Assert.ThatBool(
	actual := _List.Empty,
	message := "Clear with release must empty the list"
).IsTrue();

IF _UseDynamicStorage THEN
	Assert.ThatBool(
		actual := _List.Capacity = 0 AND_THEN GetBufferAddress() = TOF_Core.Memory.NULL_ADDRESS,
		message := "Clear with release must drop the dynamic allocation"
	).IsTrue();
ELSE
	Assert.ThatBool(
		actual := _List.Capacity = 12 AND_THEN GetBufferAddress() = buffer,
		message := "Clear with release must preserve the inline allocation"
	).IsTrue();
END_IF
END_METHOD

//! <summary>Borrows the concrete class name. Callers must not modify it.</summary>
{attribute 'monitoring' := 'call'}
PROPERTY ClassName : REFERENCE TO STRING
GET
ClassName REF= _ClassName;
END_GET
END_PROPERTY

//! <summary>Borrows the compiler-initialized namespace name. Callers must not modify it.</summary>
{attribute 'monitoring' := 'call'}
PROPERTY NamespaceName : REFERENCE TO STRING
GET
NamespaceName REF= CurrentNamespace.Name;
END_GET
END_PROPERTY

//! <summary>Reports the concrete instance size in bytes.</summary>
{attribute 'monitoring' := 'call'}
PROPERTY SelfSize : ULINT
GET
SelfSize := XSIZEOF(THIS^);
END_GET
END_PROPERTY

END_FUNCTION_BLOCK

// ---- Tests/Collections/Static/StaticByteListTestGroup.TcPOU
(*
SPDX-FileCopyrightText: c 2026 Oleksandr Tiutyk <trofimich@gmail.com>
SPDX-License-Identifier: MIT
License: https://opensource.org/license/mit
*)

(*!
<summary>Groups fixed-capacity byte-list operations and overflow handling.</summary>
<description>
Owns the independent child instances and their fixed registration array. Use from one PLC task at a stable address.
</description>
*)

{attribute 'no_assign'}
{attribute 'no_explicit_call' := 'do not call this function block directly'}
FUNCTION_BLOCK StaticByteListTestGroup EXTENDS TOF_Testing.TestGroup<7>
VAR_STAT
	{attribute 'hide'}
	_ClassName : STRING := __POUNAME();
END_VAR
VAR
	_LoadFromAny : ByteListLoadFromAnyTest(name := "LoadFromAny", parent := THIS^, useDynamicStorage := FALSE);
	_GetAndSet : ByteListIndexedAccessTest(name := "GetAndSet", parent := THIS^, useDynamicStorage := FALSE);
	_Find : ByteListFindTest(name := "Find", parent := THIS^, useDynamicStorage := FALSE);
	_Remove : ByteListRemoveValueTest(name := "Remove", parent := THIS^, useDynamicStorage := FALSE);
	_RemoveAt : ByteListRemoveRangeTest(name := "RemoveAt", parent := THIS^, useDynamicStorage := FALSE);
	_Clear : ByteListClearTest(name := "Clear", parent := THIS^, useDynamicStorage := FALSE);
	_Overflow : StaticByteListOverflowTest(name := "Overflow", parent := THIS^);

	_Children : ARRAY [0.._ChildCount - 1] OF TOF_Testing.ITestElement :=
	[
		_LoadFromAny,
		_GetAndSet,
		_Find,
		_Remove,
		_RemoveAt,
		_Clear,
		_Overflow
	];
END_VAR

//! <summary>Borrows the fixed child array. Callers must not modify it.</summary>
{attribute 'monitoring' := 'call'}
PROPERTY Children : REFERENCE TO ARRAY [0.._ChildCount - 1] OF TOF_Testing.ITestElement
GET
Children REF= _Children;
END_GET
END_PROPERTY

//! <summary>Borrows the concrete class name. Callers must not modify it.</summary>
{attribute 'monitoring' := 'call'}
PROPERTY ClassName : REFERENCE TO STRING
GET
ClassName REF= _ClassName;
END_GET
END_PROPERTY

//! <summary>Borrows the compiler-initialized namespace name. Callers must not modify it.</summary>
{attribute 'monitoring' := 'call'}
PROPERTY NamespaceName : REFERENCE TO STRING
GET
NamespaceName REF= CurrentNamespace.Name;
END_GET
END_PROPERTY

//! <summary>Reports the concrete instance size in bytes.</summary>
{attribute 'monitoring' := 'call'}
PROPERTY SelfSize : ULINT
GET
SelfSize := XSIZEOF(THIS^);
END_GET
END_PROPERTY

END_FUNCTION_BLOCK

// ---- Tests/Collections/Static/StaticByteListOverflowTest.TcPOU
(*
SPDX-FileCopyrightText: c 2026 Oleksandr Tiutyk <trofimich@gmail.com>
SPDX-License-Identifier: MIT
License: https://opensource.org/license/mit
*)

(*!
<summary>Checks full-capacity rejection, unchanged bytes and subsequent reuse.</summary>
<description>
Owns a fixed-capacity byte list. Run from one task at a stable address. Teardown clears the logical bytes.
</description>
*)

{attribute 'no_assign'}
{attribute 'no_explicit_call' := 'do not call this function block directly'}
FUNCTION_BLOCK StaticByteListOverflowTest EXTENDS TOF_Testing.SingleCycleTest
VAR_STAT
	{attribute 'hide'}
	_ClassName : STRING := __POUNAME();
END_VAR
VAR
	_List : TOF_Collections.ByteList<12>;
END_VAR

(*!
<summary>Checks full-capacity rejection, unchanged bytes and subsequent reuse.</summary>
*)
METHOD PROTECTED ExecuteTest
VAR
	values : ARRAY [0..11] OF BYTE := [1, 2, 3, 4, 5, 6, 7, 8, 9, 10, 11, 12];
	i : DINT;

	exceptionCode : __SYSTEM.ExceptionCode;
	caught : TOF_Core.IException;
	fullException : TOF_Core.IStaticCollectionFullException;
END_VAR
_List.AppendAny(data := values);

Assert.ThatBool(
	actual := _List.Full AND_THEN _List.Length = 12 AND_THEN _List.Capacity = 12,
	message := "The list must accept exactly twelve bytes"
).IsTrue();

__TRY
	_List.AppendByte(value := BYTE#255);
__CATCH(exceptionCode)
	caught := TOF_Core.ExceptionManager.GetLastException(
		exceptionCode := exceptionCode,
		catchPointNamespaceName := NamespaceName,
		catchPointPOUName := __POUNAME(),
		catchPointPosition := __POSITION()
	);
__ENDTRY

Assert.ThatBool(
	actual := __QUERYINTERFACE(caught, fullException),
	message := "Appending to a full list must raise StaticCollectionFullException"
).IsTrue();

Assert.ThatBool(
	actual := _List.Full AND_THEN _List.Length = 12 AND_THEN _List.Capacity = 12,
	message := "Rejected append must preserve the full list and its capacity"
).IsTrue();

FOR i := 0 TO 11 DO
	Assert.ThatByte(
		actual := _List.Get(index := i),
		message := "Rejected append must preserve every byte"
	).ToBe(expected := values[i]);
END_FOR

_List.RemoveAt(index := 11, count := 1);
_List.AppendByte(value := BYTE#255);

Assert.ThatBool(
	actual := _List.Full AND_THEN _List.Get(index := 11) = BYTE#255,
	message := "Freeing one slot must allow the next append"
).IsTrue();
END_METHOD

(*!
<summary>Restores the fixture before the runner publishes the result.</summary>
<description>
Also runs after an unexpected exception interrupts the case.
</description>
*)
METHOD PROTECTED AfterTest
_List.Clear(releaseDynamicMemory := TRUE);
END_METHOD

//! <summary>Borrows the concrete class name. Callers must not modify it.</summary>
{attribute 'monitoring' := 'call'}
PROPERTY ClassName : REFERENCE TO STRING
GET
ClassName REF= _ClassName;
END_GET
END_PROPERTY

//! <summary>Borrows the compiler-initialized namespace name. Callers must not modify it.</summary>
{attribute 'monitoring' := 'call'}
PROPERTY NamespaceName : REFERENCE TO STRING
GET
NamespaceName REF= CurrentNamespace.Name;
END_GET
END_PROPERTY

//! <summary>Reports the concrete instance size in bytes.</summary>
{attribute 'monitoring' := 'call'}
PROPERTY SelfSize : ULINT
GET
SelfSize := XSIZEOF(THIS^);
END_GET
END_PROPERTY

END_FUNCTION_BLOCK

// ---- Tests/JSON/AutomaticJsonSerializerTestGroup.TcPOU
(*
SPDX-FileCopyrightText: c 2026 Oleksandr Tiutyk <trofimich@gmail.com>
SPDX-License-Identifier: MIT
License: https://opensource.org/license/mit
*)

(*!
<summary>Groups native JSON conversion, capacity, encoding and callback cases.</summary>
<description>
Owns the independent child instances and their fixed registration array. Use from one PLC task at a stable address.
</description>
*)

{attribute 'no_assign'}
{attribute 'no_explicit_call' := 'do not call this function block directly'}
FUNCTION_BLOCK AutomaticJsonSerializerTestGroup EXTENDS TOF_Testing.TestGroup<12>
VAR_STAT
	{attribute 'hide'}
	_ClassName : STRING := __POUNAME();
END_VAR
VAR
	_RoundTripsAnyStructure : AutomaticJsonRoundTripsAnyStructureTest(name := "RoundTripsAnyStructure", parent := THIS^);
	_ThrowingAnyRoundTrip : AutomaticJsonThrowingAnyRoundTripTest(name := "ThrowingAnyRoundTrip", parent := THIS^);
	_SingleFieldVarInfoRoundTrip : AutomaticJsonSingleFieldVarInfoRoundTripTest(name := "SingleFieldVarInfoRoundTrip", parent := THIS^);
	_RejectsInvalidArguments : AutomaticJsonRejectsInvalidArgumentsTest(name := "RejectsInvalidArguments", parent := THIS^);
	_ThrowingArgumentCategories : AutomaticJsonThrowingArgumentCategoriesTest(name := "ThrowingArgumentCategories", parent := THIS^);
	_MalformedJsonAndReuse : AutomaticJsonMalformedJsonAndReuseTest(name := "MalformedJsonAndReuse", parent := THIS^);
	_WrappedCallbacks : AutomaticJsonWrappedCallbacksTest(name := "WrappedCallbacks", parent := THIS^);
	_CallbackContainmentAndReuse : AutomaticJsonCallbackContainmentAndReuseTest(name := "CallbackContainmentAndReuse", parent := THIS^);
	_ThrowingCallbackPropagation : AutomaticJsonThrowingCallbackPropagationTest(name := "ThrowingCallbackPropagation", parent := THIS^);
	_CapacityOverflowAndReuse : AutomaticJsonCapacityOverflowAndReuseTest(name := "CapacityOverflowAndReuse", parent := THIS^);
	_LongUtf8RoundTrip : AutomaticJsonLongUtf8RoundTripTest(name := "LongUtf8RoundTrip", parent := THIS^);
	_DecimalPlacesReadback : AutomaticJsonDecimalPlacesReadbackTest(name := "DecimalPlacesReadback", parent := THIS^);

	_Children : ARRAY [0.._ChildCount - 1] OF TOF_Testing.ITestElement :=
	[
		_RoundTripsAnyStructure,
		_ThrowingAnyRoundTrip,
		_SingleFieldVarInfoRoundTrip,
		_RejectsInvalidArguments,
		_ThrowingArgumentCategories,
		_MalformedJsonAndReuse,
		_WrappedCallbacks,
		_CallbackContainmentAndReuse,
		_ThrowingCallbackPropagation,
		_CapacityOverflowAndReuse,
		_LongUtf8RoundTrip,
		_DecimalPlacesReadback
	];
END_VAR

//! <summary>Borrows the fixed child array. Callers must not modify it.</summary>
{attribute 'monitoring' := 'call'}
PROPERTY Children : REFERENCE TO ARRAY [0.._ChildCount - 1] OF TOF_Testing.ITestElement
GET
Children REF= _Children;
END_GET
END_PROPERTY

//! <summary>Borrows the concrete class name. Callers must not modify it.</summary>
{attribute 'monitoring' := 'call'}
PROPERTY ClassName : REFERENCE TO STRING
GET
ClassName REF= _ClassName;
END_GET
END_PROPERTY

//! <summary>Borrows the compiler-initialized namespace name. Callers must not modify it.</summary>
{attribute 'monitoring' := 'call'}
PROPERTY NamespaceName : REFERENCE TO STRING
GET
NamespaceName REF= CurrentNamespace.Name;
END_GET
END_PROPERTY

//! <summary>Reports the concrete instance size in bytes.</summary>
{attribute 'monitoring' := 'call'}
PROPERTY SelfSize : ULINT
GET
SelfSize := XSIZEOF(THIS^);
END_GET
END_PROPERTY

END_FUNCTION_BLOCK

// ---- Tests/JSON/AutomaticJsonRoundTripsAnyStructureTest.TcPOU
(*
SPDX-FileCopyrightText: c 2026 Oleksandr Tiutyk <trofimich@gmail.com>
SPDX-License-Identifier: MIT
License: https://opensource.org/license/mit
*)

(*!
<summary>Checks successful ANY Try conversion and copied byte count.</summary>
<description>
Owns persistent native serializer state and any payload buffers used by this case.
Run from one task at a stable address. The caller provides task-boundary exception cleanup.
</description>
*)

{attribute 'no_assign'}
{attribute 'no_explicit_call' := 'do not call this function block directly'}
FUNCTION_BLOCK AutomaticJsonRoundTripsAnyStructureTest EXTENDS TOF_Testing.SingleCycleTest
VAR_STAT
	{attribute 'hide'}
	_ClassName : STRING := __POUNAME();
END_VAR
VAR
	_Serializer : TOF_JSON.AutomaticJsonSerializer;
	_Source : JSON_TEST_VALUE;
	_Target : JSON_TEST_VALUE;
	_Json : TOF_Core.JSON_DOCUMENT;
END_VAR

(*!
<summary>Checks successful ANY Try conversion and copied byte count.</summary>
*)
METHOD PROTECTED ExecuteTest
VAR
	success : BOOL;
	jsonSize : UDINT;
	expectedJson : STRING(40) := '{"Number":42,"Ready":true}';
END_VAR
_Source.Number := 42;
_Source.Ready := TRUE;

_Target.Number := 0;
_Target.Ready := FALSE;

_Json := '';

success := _Serializer.TrySerialize(
	sourceStructure := _Source,
	extender := 0,
	targetJson := _Json,
	jsonSize => jsonSize
);
Assert.ThatBool(
	actual := success,
	message := "ANY TryCreate must succeed"
).IsTrue();
Assert.ThatUDInt(
	actual := jsonSize,
	message := "Copy count must include the terminator"
).ToBe(expected := TOF_Core.Strings.GetLength(value := _Json) + 1);

Assert.That(
	actual := _Json,
	message := "Serialization must emit the expected structure members"
).ToBe(expected := expectedJson);

success := _Serializer.TryDeserialize(json := _Json, targetStructure := _Target);
Assert.ThatBool(
	actual := success,
	message := "ANY TryFill must succeed"
).IsTrue();
Assert.ThatDInt(
	actual := _Target.Number,
	message := "Integer payload must round-trip"
).ToBe(expected := 42);
Assert.ThatBool(
	actual := _Target.Ready,
	message := "Boolean payload must round-trip"
).IsTrue();
END_METHOD

//! <summary>Borrows the concrete class name. Callers must not modify it.</summary>
{attribute 'monitoring' := 'call'}
PROPERTY ClassName : REFERENCE TO STRING
GET
ClassName REF= _ClassName;
END_GET
END_PROPERTY

//! <summary>Borrows the compiler-initialized namespace name. Callers must not modify it.</summary>
{attribute 'monitoring' := 'call'}
PROPERTY NamespaceName : REFERENCE TO STRING
GET
NamespaceName REF= CurrentNamespace.Name;
END_GET
END_PROPERTY

//! <summary>Reports the concrete instance size in bytes.</summary>
{attribute 'monitoring' := 'call'}
PROPERTY SelfSize : ULINT
GET
SelfSize := XSIZEOF(THIS^);
END_GET
END_PROPERTY

END_FUNCTION_BLOCK

// ---- Tests/JSON/AutomaticJsonThrowingAnyRoundTripTest.TcPOU
(*
SPDX-FileCopyrightText: c 2026 Oleksandr Tiutyk <trofimich@gmail.com>
SPDX-License-Identifier: MIT
License: https://opensource.org/license/mit
*)

(*!
<summary>Checks successful throwing ANY serialization and restoration.</summary>
<description>
Owns persistent native serializer state and any payload buffers used by this case.
Run from one task at a stable address. The caller provides task-boundary exception cleanup.
</description>
*)

{attribute 'no_assign'}
{attribute 'no_explicit_call' := 'do not call this function block directly'}
FUNCTION_BLOCK AutomaticJsonThrowingAnyRoundTripTest EXTENDS TOF_Testing.SingleCycleTest
VAR_STAT
	{attribute 'hide'}
	_ClassName : STRING := __POUNAME();
END_VAR
VAR
	_Serializer : TOF_JSON.AutomaticJsonSerializer;
	_Source : JSON_TEST_VALUE;
	_Target : JSON_TEST_VALUE;
	_Json : TOF_Core.JSON_DOCUMENT;
END_VAR

(*!
<summary>Checks successful throwing ANY serialization and restoration.</summary>
*)
METHOD PROTECTED ExecuteTest
VAR
	jsonSize : UDINT;
	expectedJson : STRING(40) := '{"Number":42,"Ready":true}';
END_VAR
_Source.Number := 42;
_Source.Ready := TRUE;

_Target.Number := 0;
_Target.Ready := FALSE;

_Json := '';

_Serializer.Serialize(
	sourceStructure := _Source,
	extender := 0,
	targetJson := _Json,
	jsonSize => jsonSize
);

Assert.That(
	actual := _Json,
	message := "Serialization must emit the expected structure members"
).ToBe(expected := expectedJson);

_Serializer.Deserialize(json := _Json, targetStructure := _Target);
Assert.ThatDInt(
	actual := _Target.Number,
	message := "Integer payload must round-trip"
).ToBe(expected := 42);
Assert.ThatBool(
	actual := _Target.Ready,
	message := "Boolean payload must round-trip"
).IsTrue();
END_METHOD

//! <summary>Borrows the concrete class name. Callers must not modify it.</summary>
{attribute 'monitoring' := 'call'}
PROPERTY ClassName : REFERENCE TO STRING
GET
ClassName REF= _ClassName;
END_GET
END_PROPERTY

//! <summary>Borrows the compiler-initialized namespace name. Callers must not modify it.</summary>
{attribute 'monitoring' := 'call'}
PROPERTY NamespaceName : REFERENCE TO STRING
GET
NamespaceName REF= CurrentNamespace.Name;
END_GET
END_PROPERTY

//! <summary>Reports the concrete instance size in bytes.</summary>
{attribute 'monitoring' := 'call'}
PROPERTY SelfSize : ULINT
GET
SelfSize := XSIZEOF(THIS^);
END_GET
END_PROPERTY

END_FUNCTION_BLOCK

// ---- Tests/JSON/AutomaticJsonSingleFieldVarInfoRoundTripTest.TcPOU
(*
SPDX-FileCopyrightText: c 2026 Oleksandr Tiutyk <trofimich@gmail.com>
SPDX-License-Identifier: MIT
License: https://opensource.org/license/mit
*)

(*!
<summary>Checks both throwing and Try VAR_INFO paths for a single-field structure.</summary>
<description>
Owns persistent native serializer state and any payload buffers used by this case.
Run from one task at a stable address. The caller provides task-boundary exception cleanup.
</description>
*)

{attribute 'no_assign'}
{attribute 'no_explicit_call' := 'do not call this function block directly'}
FUNCTION_BLOCK AutomaticJsonSingleFieldVarInfoRoundTripTest EXTENDS TOF_Testing.SingleCycleTest
VAR_STAT
	{attribute 'hide'}
	_ClassName : STRING := __POUNAME();
END_VAR
VAR
	_Serializer : TOF_JSON.AutomaticJsonSerializer;
	_SingleSource : JSON_TEST_SINGLE_VALUE;
	_SingleTarget : JSON_TEST_SINGLE_VALUE;
	_Json : TOF_Core.JSON_DOCUMENT;
END_VAR

(*!
<summary>Checks both throwing and Try VAR_INFO paths for a single-field structure.</summary>
*)
METHOD PROTECTED ExecuteTest
VAR
	sourceInfo : __SYSTEM.VAR_INFO;
	targetInfo : __SYSTEM.VAR_INFO;
	success : BOOL;
	jsonSize : UDINT;
END_VAR
_Json := '';

_SingleSource.Number := -17;
_SingleTarget.Number := 0;
sourceInfo := __VARINFO(_SingleSource);
targetInfo := __VARINFO(_SingleTarget);
// Regression: explicit pointers must drive all four paths when descriptor addresses are absent.
sourceInfo.ByteAddress := TOF_Core.UnsignedInt32.ZERO;
targetInfo.ByteAddress := TOF_Core.UnsignedInt32.ZERO;
success := _Serializer.TrySerializeByVarInfo(
	sourceStructureVarInfo := sourceInfo,
	sourceStructureAddress := ADR(_SingleSource),
	extender := 0,
	targetJson := _Json,
	jsonSize => jsonSize
);
Assert.ThatBool(
	actual := success,
	message := "Explicit single-field TryCreate must succeed"
).IsTrue();
_Serializer.DeserializeByVarInfo(
	json := _Json,
	targetStructureVarInfo := targetInfo,
	targetStructureAddress := ADR(_SingleTarget)
);
Assert.ThatDInt(
	actual := _SingleTarget.Number,
	message := "Explicit type must restore the structure"
).ToBe(expected := -17);
_SingleSource.Number := 91;
_Serializer.SerializeByVarInfo(
	sourceStructureVarInfo := sourceInfo,
	sourceStructureAddress := ADR(_SingleSource),
	extender := 0,
	targetJson := _Json,
	jsonSize => jsonSize
);
success := _Serializer.TryDeserializeByVarInfo(
	json := _Json,
	targetStructureVarInfo := targetInfo,
	targetStructureAddress := ADR(_SingleTarget)
);
Assert.ThatBool(
	actual := success,
	message := "Explicit single-field TryFill must succeed"
).IsTrue();
Assert.ThatDInt(
	actual := _SingleTarget.Number,
	message := "Try must use the supplied type"
).ToBe(expected := 91);
END_METHOD

//! <summary>Borrows the concrete class name. Callers must not modify it.</summary>
{attribute 'monitoring' := 'call'}
PROPERTY ClassName : REFERENCE TO STRING
GET
ClassName REF= _ClassName;
END_GET
END_PROPERTY

//! <summary>Borrows the compiler-initialized namespace name. Callers must not modify it.</summary>
{attribute 'monitoring' := 'call'}
PROPERTY NamespaceName : REFERENCE TO STRING
GET
NamespaceName REF= CurrentNamespace.Name;
END_GET
END_PROPERTY

//! <summary>Reports the concrete instance size in bytes.</summary>
{attribute 'monitoring' := 'call'}
PROPERTY SelfSize : ULINT
GET
SelfSize := XSIZEOF(THIS^);
END_GET
END_PROPERTY

END_FUNCTION_BLOCK

// ---- Tests/JSON/AutomaticJsonRejectsInvalidArgumentsTest.TcPOU
(*
SPDX-FileCopyrightText: c 2026 Oleksandr Tiutyk <trofimich@gmail.com>
SPDX-License-Identifier: MIT
License: https://opensource.org/license/mit
*)

(*!
<summary>Checks ordinary Try refusals without leaking exceptions or invoking hooks.</summary>
<description>
Owns persistent native serializer state and any payload buffers used by this case.
Run from one task at a stable address. The caller provides task-boundary exception cleanup.
</description>
*)

{attribute 'no_assign'}
{attribute 'no_explicit_call' := 'do not call this function block directly'}
FUNCTION_BLOCK AutomaticJsonRejectsInvalidArgumentsTest EXTENDS TOF_Testing.SingleCycleTest
VAR_STAT
	{attribute 'hide'}
	_ClassName : STRING := __POUNAME();
END_VAR
VAR
	_Serializer : TOF_JSON.AutomaticJsonSerializer;
	_Extender : JsonExtenderProbe;
	_Source : JSON_TEST_VALUE;
	_Json : TOF_Core.JSON_DOCUMENT;
END_VAR

(*!
<summary>Checks ordinary Try refusals without leaking exceptions or invoking hooks.</summary>
*)
METHOD PROTECTED ExecuteTest
VAR
	scalar : DINT;
	structureAddress : PVOID;
	sourceInfo : __SYSTEM.VAR_INFO;
	success : BOOL;
	jsonSize : UDINT;
	leaked : BOOL;
END_VAR
_Source.Number := 42;
_Source.Ready := TRUE;

_Json := '';

_Extender.Reset();

scalar := 3;
_Json := '{"Number":42,"Ready":true}';

__TRY
	success := _Serializer.TrySerialize(
		sourceStructure := scalar,
		extender := _Extender,
		targetJson := _Json,
		jsonSize => jsonSize
	);
	Assert.ThatBool(
		actual := success,
		message := "Scalar ANY must be rejected"
	).IsFalse();
	success := _Serializer.TryDeserialize(json := _Json, targetStructure := scalar);
	Assert.ThatBool(
		actual := success,
		message := "Scalar ANY destination must be rejected"
	).IsFalse();
	sourceInfo := __VARINFO(scalar);
	structureAddress := ADR(scalar);
	success := _Serializer.TrySerializeByVarInfo(
		sourceStructureVarInfo := sourceInfo,
		sourceStructureAddress := structureAddress,
		extender := _Extender,
		targetJson := _Json,
		jsonSize => jsonSize
	);
	Assert.ThatBool(
		actual := success,
		message := "Scalar descriptor must be rejected"
	).IsFalse();
	success := _Serializer.TryDeserializeByVarInfo(
		json := _Json,
		targetStructureVarInfo := sourceInfo,
		targetStructureAddress := structureAddress
	);
	Assert.ThatBool(
		actual := success,
		message := "Scalar descriptor destination must be rejected"
	).IsFalse();
	sourceInfo := __VARINFO(_Source);
	structureAddress := TOF_Core.Memory.NULL_ADDRESS;
	success := _Serializer.TrySerializeByVarInfo(
		sourceStructureVarInfo := sourceInfo,
		sourceStructureAddress := structureAddress,
		extender := _Extender,
		targetJson := _Json,
		jsonSize => jsonSize
	);
	Assert.ThatBool(
		actual := success,
		message := "Null source address must be rejected"
	).IsFalse();
	success := _Serializer.TryDeserializeByVarInfo(
		json := _Json,
		targetStructureVarInfo := sourceInfo,
		targetStructureAddress := structureAddress
	);
	Assert.ThatBool(
		actual := success,
		message := "Null destination address must be rejected"
	).IsFalse();
__CATCH
	leaked := TRUE;
__ENDTRY

Assert.ThatBool(
	actual := leaked,
	message := "Try argument failures must not escape"
).IsFalse();
Assert.ThatUDInt(
	actual := _Extender.StartCount,
	message := "Rejected arguments must skip start"
).ToBe(expected := 0);
Assert.ThatUDInt(
	actual := _Extender.FinishCount,
	message := "Rejected arguments must skip finish"
).ToBe(expected := 0);
END_METHOD

(*!
<summary>Restores the fixture before the runner publishes the result.</summary>
<description>
Also runs after an unexpected exception interrupts the case.
</description>
*)
METHOD PROTECTED AfterTest
_Extender.Reset();
END_METHOD

//! <summary>Borrows the concrete class name. Callers must not modify it.</summary>
{attribute 'monitoring' := 'call'}
PROPERTY ClassName : REFERENCE TO STRING
GET
ClassName REF= _ClassName;
END_GET
END_PROPERTY

//! <summary>Borrows the compiler-initialized namespace name. Callers must not modify it.</summary>
{attribute 'monitoring' := 'call'}
PROPERTY NamespaceName : REFERENCE TO STRING
GET
NamespaceName REF= CurrentNamespace.Name;
END_GET
END_PROPERTY

//! <summary>Reports the concrete instance size in bytes.</summary>
{attribute 'monitoring' := 'call'}
PROPERTY SelfSize : ULINT
GET
SelfSize := XSIZEOF(THIS^);
END_GET
END_PROPERTY

END_FUNCTION_BLOCK

// ---- Tests/JSON/JsonExtenderProbe.TcPOU
(*
SPDX-FileCopyrightText: © 2026 Oleksandr Tiutyk <trofimich@gmail.com>
SPDX-License-Identifier: MIT
License: https://opensource.org/license/mit
*)

(*!
<summary>Wraps the structure in an array and injects recoverable callback exceptions.</summary>
<description>
Used only by the owner task of the serializer under test. Does not retain the borrowed writer or raise
terminal allocation failures; such failures require isolated owner verification.
</description>
*)

FUNCTION_BLOCK JsonExtenderProbe EXTENDS TOF_Core.Object IMPLEMENTS TOF_JSON.IJsonExtender
VAR_INPUT
	//! <summary>Raises a framework exception before writing the array prefix.</summary>
	ThrowAtStart : BOOL;
	//! <summary>Raises a framework exception before writing the array suffix.</summary>
	ThrowAtFinish : BOOL;
END_VAR
VAR_OUTPUT
	//! <summary>Observed start hooks since Reset.</summary>
	StartCount : UDINT;
	//! <summary>Observed finish hooks since Reset.</summary>
	FinishCount : UDINT;
END_VAR
VAR_STAT
	_ClassName : STRING := __POUNAME();
END_VAR

(*!
<summary>Borrows the immutable fixture class name for its lifetime.</summary>
*)
PROPERTY ClassName : REFERENCE TO STRING
GET
ClassName REF= _ClassName;
END_GET
END_PROPERTY

(*!
<summary>Borrows read-only compiler-initialized test namespace storage.</summary>
*)
PROPERTY NamespaceName : REFERENCE TO STRING
GET
NamespaceName REF= CurrentNamespace.Name;
END_GET
END_PROPERTY

(*!
<summary>Reports the complete fixture instance size in bytes.</summary>
*)
PROPERTY SelfSize : ULINT
GET
SelfSize := XSIZEOF(THIS^);
END_GET
END_PROPERTY

(*!
<summary>Clears callback observations and disables both exception injections.</summary>
*)
METHOD Reset
StartCount := TOF_Core.UnsignedInt32.ZERO;
FinishCount := TOF_Core.UnsignedInt32.ZERO;
ThrowAtStart := FALSE;
ThrowAtFinish := FALSE;
END_METHOD

(*!
<summary>Counts this hook and writes its array boundary unless configured to raise.</summary>
<description>
Borrows the writer only for this synchronous call and retains no reference. Native failures raise a
framework exception so the serializer can exercise its throwing or Try boundary.
</description>
*)
//! <param name="jsonSaxWriter">Borrowed writer owned by the active serializer.</param>
METHOD WritePrefix
VAR_IN_OUT CONSTANT
	jsonSaxWriter : Tc3_JsonXml.FB_JsonSaxWriter;
END_VAR
VAR
	errorCode : HRESULT;
END_VAR
StartCount := StartCount + 1;

IF ThrowAtStart THEN
	TOF_Core.Exceptions.ThrowStandard(
		sourceNamespaceName := NamespaceName,
		sourceClassName := ClassName,
		sourcePOUName := __POUNAME(),
		sourcePosition := __POSITION(),
		message := "JSON extender injected failure"
	);
END_IF

errorCode := jsonSaxWriter.StartArray();

IF errorCode <> TOF_Core.SignedInt32.ZERO THEN
	TOF_Core.Exceptions.ThrowStandard(
		sourceNamespaceName := NamespaceName,
		sourceClassName := ClassName,
		sourcePOUName := __POUNAME(),
		sourcePosition := __POSITION(),
		message := "JSON extender could not write its array boundary",
		errorCode := TO_UDINT(errorCode)
	);
END_IF
END_METHOD

(*!
<summary>Counts this hook and writes its array boundary unless configured to raise.</summary>
<description>
Borrows the writer only for this synchronous call and retains no reference. Native failures raise a
framework exception so the serializer can exercise its throwing or Try boundary.
</description>
*)
//! <param name="jsonSaxWriter">Borrowed writer owned by the active serializer.</param>
METHOD WriteSuffix
VAR_IN_OUT CONSTANT
	jsonSaxWriter : Tc3_JsonXml.FB_JsonSaxWriter;
END_VAR
VAR
	errorCode : HRESULT;
END_VAR
FinishCount := FinishCount + 1;

IF ThrowAtFinish THEN
	TOF_Core.Exceptions.ThrowStandard(
		sourceNamespaceName := NamespaceName,
		sourceClassName := ClassName,
		sourcePOUName := __POUNAME(),
		sourcePosition := __POSITION(),
		message := "JSON extender injected failure"
	);
END_IF

errorCode := jsonSaxWriter.EndArray();

IF errorCode <> TOF_Core.SignedInt32.ZERO THEN
	TOF_Core.Exceptions.ThrowStandard(
		sourceNamespaceName := NamespaceName,
		sourceClassName := ClassName,
		sourcePOUName := __POUNAME(),
		sourcePosition := __POSITION(),
		message := "JSON extender could not write its array boundary",
		errorCode := TO_UDINT(errorCode)
	);
END_IF
END_METHOD

END_FUNCTION_BLOCK

// ---- Tests/JSON/AutomaticJsonThrowingArgumentCategoriesTest.TcPOU
(*
SPDX-FileCopyrightText: c 2026 Oleksandr Tiutyk <trofimich@gmail.com>
SPDX-License-Identifier: MIT
License: https://opensource.org/license/mit
*)

(*!
<summary>Checks null source and target addresses and unsupported-type exception categories.</summary>
<description>
Owns persistent native serializer state and any payload buffers used by this case.
Run from one task at a stable address. The caller provides task-boundary exception cleanup.
</description>
*)

{attribute 'no_assign'}
{attribute 'no_explicit_call' := 'do not call this function block directly'}
FUNCTION_BLOCK AutomaticJsonThrowingArgumentCategoriesTest EXTENDS TOF_Testing.SingleCycleTest
VAR_STAT
	{attribute 'hide'}
	_ClassName : STRING := __POUNAME();
END_VAR
VAR
	_Serializer : TOF_JSON.AutomaticJsonSerializer;
	_Source : JSON_TEST_VALUE;
	_Json : TOF_Core.JSON_DOCUMENT;
END_VAR

(*!
<summary>Checks null source and target addresses and unsupported-type exception categories.</summary>
*)
METHOD PROTECTED ExecuteTest
VAR
	caught : BOOL;
	exceptionCode : __SYSTEM.ExceptionCode;
	caughtException : TOF_Core.IException;
	scalar : DINT;
	sourceInfo : __SYSTEM.VAR_INFO;
	jsonSize : UDINT;
	missing : TOF_Core.IArgumentNotSpecifiedException;
	unsupported : TOF_Core.IArgumentTypeClassNotSupportedException;
END_VAR
_Source.Number := 42;
_Source.Ready := TRUE;

_Json := '';

sourceInfo := __VARINFO(_Source);
sourceInfo.ByteAddress := TOF_Core.UnsignedInt32.ZERO;

__TRY
	_Serializer.SerializeByVarInfo(
		sourceStructureVarInfo := sourceInfo,
		sourceStructureAddress := TOF_Core.Memory.NULL_ADDRESS,
		extender := 0,
		targetJson := _Json,
		jsonSize => jsonSize
	);
__CATCH(exceptionCode)
	caught := TRUE;
	caughtException := TOF_Core.ExceptionManager.GetLastException(
		exceptionCode := exceptionCode,
		catchPointNamespaceName := CurrentNamespace.Name,
		catchPointPOUName := __POUNAME(),
		catchPointPosition := __POSITION()
	);
	Assert.ThatBool(
		actual := __QUERYINTERFACE(caughtException, missing),
		message := "Null source must retain the required-argument category"
	).IsTrue();
__ENDTRY

Assert.ThatBool(
	actual := caught,
	message := "Throwing API must reject a null source"
).IsTrue();
caught := FALSE;

// Verify the address guard without entering native conversion.
__TRY
	_Serializer.DeserializeByVarInfo(
		json := _Json,
		targetStructureVarInfo := sourceInfo,
		targetStructureAddress := TOF_Core.Memory.NULL_ADDRESS
	);
__CATCH(exceptionCode)
	caught := TRUE;
	caughtException := TOF_Core.ExceptionManager.GetLastException(
		exceptionCode := exceptionCode,
		catchPointNamespaceName := CurrentNamespace.Name,
		catchPointPOUName := __POUNAME(),
		catchPointPosition := __POSITION()
	);
	Assert.ThatBool(
		actual := __QUERYINTERFACE(caughtException, missing),
		message := "Null target must retain the required-argument category"
	).IsTrue();
__ENDTRY

Assert.ThatBool(
	actual := caught,
	message := "Throwing API must reject a null target"
).IsTrue();
caught := FALSE;

__TRY
	_Serializer.Deserialize(json := _Json, targetStructure := scalar);
__CATCH(exceptionCode)
	caught := TRUE;
	caughtException := TOF_Core.ExceptionManager.GetLastException(
		exceptionCode := exceptionCode,
		catchPointNamespaceName := CurrentNamespace.Name,
		catchPointPOUName := __POUNAME(),
		catchPointPosition := __POSITION()
	);
	Assert.ThatBool(
		actual := __QUERYINTERFACE(caughtException, unsupported),
		message := "Scalar target must retain the unsupported-type category"
	).IsTrue();
__ENDTRY

Assert.ThatBool(
	actual := caught,
	message := "Throwing API must reject a scalar target"
).IsTrue();
END_METHOD

//! <summary>Borrows the concrete class name. Callers must not modify it.</summary>
{attribute 'monitoring' := 'call'}
PROPERTY ClassName : REFERENCE TO STRING
GET
ClassName REF= _ClassName;
END_GET
END_PROPERTY

//! <summary>Borrows the compiler-initialized namespace name. Callers must not modify it.</summary>
{attribute 'monitoring' := 'call'}
PROPERTY NamespaceName : REFERENCE TO STRING
GET
NamespaceName REF= CurrentNamespace.Name;
END_GET
END_PROPERTY

//! <summary>Reports the concrete instance size in bytes.</summary>
{attribute 'monitoring' := 'call'}
PROPERTY SelfSize : ULINT
GET
SelfSize := XSIZEOF(THIS^);
END_GET
END_PROPERTY

END_FUNCTION_BLOCK

// ---- Tests/JSON/AutomaticJsonMalformedJsonAndReuseTest.TcPOU
(*
SPDX-FileCopyrightText: c 2026 Oleksandr Tiutyk <trofimich@gmail.com>
SPDX-License-Identifier: MIT
License: https://opensource.org/license/mit
*)

(*!
<summary>Checks malformed-input refusal and successful reuse of both fill paths.</summary>
<description>
Owns persistent native serializer state and any payload buffers used by this case.
Run from one task at a stable address. The caller provides task-boundary exception cleanup.
</description>
*)

{attribute 'no_assign'}
{attribute 'no_explicit_call' := 'do not call this function block directly'}
FUNCTION_BLOCK AutomaticJsonMalformedJsonAndReuseTest EXTENDS TOF_Testing.SingleCycleTest
VAR_STAT
	{attribute 'hide'}
	_ClassName : STRING := __POUNAME();
END_VAR
VAR
	_Serializer : TOF_JSON.AutomaticJsonSerializer;
	_Target : JSON_TEST_VALUE;
	_Json : TOF_Core.JSON_DOCUMENT;
END_VAR

(*!
<summary>Checks malformed-input refusal and successful reuse of both fill paths.</summary>
*)
METHOD PROTECTED ExecuteTest
VAR
	targetInfo : __SYSTEM.VAR_INFO;
	success : BOOL;
END_VAR
_Target.Number := 0;
_Target.Ready := FALSE;

_Json := '{';
targetInfo := __VARINFO(_Target);
success := _Serializer.TryDeserialize(json := _Json, targetStructure := _Target);
Assert.ThatBool(
	actual := success,
	message := "Malformed JSON must fail ANY TryFill"
).IsFalse();
success := _Serializer.TryDeserializeByVarInfo(
	json := _Json,
	targetStructureVarInfo := targetInfo,
	targetStructureAddress := ADR(_Target)
);
Assert.ThatBool(
	actual := success,
	message := "Malformed JSON must fail explicit TryFill"
).IsFalse();
_Json := '{"Number":42,"Ready":true}';
success := _Serializer.TryDeserialize(json := _Json, targetStructure := _Target);
Assert.ThatBool(
	actual := success,
	message := "ANY fill must recover on the next valid call"
).IsTrue();
Assert.ThatDInt(
	actual := _Target.Number,
	message := "Integer payload must round-trip"
).ToBe(expected := 42);
Assert.ThatBool(
	actual := _Target.Ready,
	message := "Boolean payload must round-trip"
).IsTrue();
_Target.Number := 0;
_Target.Ready := FALSE;
success := _Serializer.TryDeserializeByVarInfo(
	json := _Json,
	targetStructureVarInfo := targetInfo,
	targetStructureAddress := ADR(_Target)
);
Assert.ThatBool(
	actual := success,
	message := "Explicit fill must recover on the next valid call"
).IsTrue();
Assert.ThatDInt(
	actual := _Target.Number,
	message := "Integer payload must round-trip"
).ToBe(expected := 42);
Assert.ThatBool(
	actual := _Target.Ready,
	message := "Boolean payload must round-trip"
).IsTrue();
END_METHOD

//! <summary>Borrows the concrete class name. Callers must not modify it.</summary>
{attribute 'monitoring' := 'call'}
PROPERTY ClassName : REFERENCE TO STRING
GET
ClassName REF= _ClassName;
END_GET
END_PROPERTY

//! <summary>Borrows the compiler-initialized namespace name. Callers must not modify it.</summary>
{attribute 'monitoring' := 'call'}
PROPERTY NamespaceName : REFERENCE TO STRING
GET
NamespaceName REF= CurrentNamespace.Name;
END_GET
END_PROPERTY

//! <summary>Reports the concrete instance size in bytes.</summary>
{attribute 'monitoring' := 'call'}
PROPERTY SelfSize : ULINT
GET
SelfSize := XSIZEOF(THIS^);
END_GET
END_PROPERTY

END_FUNCTION_BLOCK

// ---- Tests/JSON/AutomaticJsonWrappedCallbacksTest.TcPOU
(*
SPDX-FileCopyrightText: c 2026 Oleksandr Tiutyk <trofimich@gmail.com>
SPDX-License-Identifier: MIT
License: https://opensource.org/license/mit
*)

(*!
<summary>Checks prefix/value/suffix order and callback counts.</summary>
<description>
Owns persistent native serializer state and any payload buffers used by this case.
Run from one task at a stable address. The caller provides task-boundary exception cleanup.
</description>
*)

{attribute 'no_assign'}
{attribute 'no_explicit_call' := 'do not call this function block directly'}
FUNCTION_BLOCK AutomaticJsonWrappedCallbacksTest EXTENDS TOF_Testing.SingleCycleTest
VAR_STAT
	{attribute 'hide'}
	_ClassName : STRING := __POUNAME();
END_VAR
VAR
	_Serializer : TOF_JSON.AutomaticJsonSerializer;
	_Extender : JsonExtenderProbe;
	_Source : JSON_TEST_VALUE;
	_Json : TOF_Core.JSON_DOCUMENT;
END_VAR

(*!
<summary>Checks prefix/value/suffix order and callback counts.</summary>
*)
METHOD PROTECTED ExecuteTest
VAR
	success : BOOL;
	jsonSize : UDINT;
	expectedJson : STRING(40) := '[{"Number":42,"Ready":true}]';
END_VAR
_Source.Number := 42;
_Source.Ready := TRUE;

_Json := '';

_Extender.Reset();

success := _Serializer.TrySerialize(
	sourceStructure := _Source,
	extender := _Extender,
	targetJson := _Json,
	jsonSize => jsonSize
);
Assert.ThatBool(
	actual := success,
	message := "Balanced callbacks must produce a document"
).IsTrue();
Assert.That(
	actual := _Json,
	message := "Callbacks must surround exactly one structure value"
).ToBe(expected := expectedJson);
Assert.ThatUDInt(
	actual := _Extender.StartCount,
	message := "Start must run once"
).ToBe(expected := 1);
Assert.ThatUDInt(
	actual := _Extender.FinishCount,
	message := "Finish must run once"
).ToBe(expected := 1);
END_METHOD

(*!
<summary>Restores the fixture before the runner publishes the result.</summary>
<description>
Also runs after an unexpected exception interrupts the case.
</description>
*)
METHOD PROTECTED AfterTest
_Extender.Reset();
END_METHOD

//! <summary>Borrows the concrete class name. Callers must not modify it.</summary>
{attribute 'monitoring' := 'call'}
PROPERTY ClassName : REFERENCE TO STRING
GET
ClassName REF= _ClassName;
END_GET
END_PROPERTY

//! <summary>Borrows the compiler-initialized namespace name. Callers must not modify it.</summary>
{attribute 'monitoring' := 'call'}
PROPERTY NamespaceName : REFERENCE TO STRING
GET
NamespaceName REF= CurrentNamespace.Name;
END_GET
END_PROPERTY

//! <summary>Reports the concrete instance size in bytes.</summary>
{attribute 'monitoring' := 'call'}
PROPERTY SelfSize : ULINT
GET
SelfSize := XSIZEOF(THIS^);
END_GET
END_PROPERTY

END_FUNCTION_BLOCK

// ---- Tests/JSON/AutomaticJsonCallbackContainmentAndReuseTest.TcPOU
(*
SPDX-FileCopyrightText: c 2026 Oleksandr Tiutyk <trofimich@gmail.com>
SPDX-License-Identifier: MIT
License: https://opensource.org/license/mit
*)

(*!
<summary>Checks exceptions from each hook in both TryCreate paths and writer reset on reuse.</summary>
<description>
Owns persistent native serializer state and any payload buffers used by this case.
Run from one task at a stable address. The caller provides task-boundary exception cleanup.
</description>
*)

{attribute 'no_assign'}
{attribute 'no_explicit_call' := 'do not call this function block directly'}
FUNCTION_BLOCK AutomaticJsonCallbackContainmentAndReuseTest EXTENDS TOF_Testing.SingleCycleTest
VAR_STAT
	{attribute 'hide'}
	_ClassName : STRING := __POUNAME();
END_VAR
VAR
	_Serializer : TOF_JSON.AutomaticJsonSerializer;
	_Extender : JsonExtenderProbe;
	_Source : JSON_TEST_VALUE;
	_Json : TOF_Core.JSON_DOCUMENT;
END_VAR

(*!
<summary>Checks exceptions from each hook in both TryCreate paths and writer reset on reuse.</summary>
*)
METHOD PROTECTED ExecuteTest
VAR
	i : INT;
	sourceInfo : __SYSTEM.VAR_INFO;
	success : BOOL;
	leaked : BOOL;
	jsonSize : UDINT;
	expectedJson : STRING(40) := '[{"Number":42,"Ready":true}]';
END_VAR
_Source.Number := 42;
_Source.Ready := TRUE;

_Json := '';

_Extender.Reset();

sourceInfo := __VARINFO(_Source);

FOR i := 0 TO 3 DO
	_Extender.Reset();
	_Extender.ThrowAtStart := (i MOD 2) = 0;
	_Extender.ThrowAtFinish := NOT _Extender.ThrowAtStart;
	leaked := FALSE;

	__TRY
		IF i < 2 THEN
			success := _Serializer.TrySerialize(
				sourceStructure := _Source,
				extender := _Extender,
				targetJson := _Json,
				jsonSize => jsonSize
			);
		ELSE
			success := _Serializer.TrySerializeByVarInfo(
				sourceStructureVarInfo := sourceInfo,
				sourceStructureAddress := ADR(_Source),
				extender := _Extender,
				targetJson := _Json,
				jsonSize => jsonSize
			);
		END_IF
	__CATCH
		leaked := TRUE;
	__ENDTRY

	Assert.ThatBool(
		actual := leaked,
		message := "Callback exception must not escape Try"
	).IsFalse();
	Assert.ThatBool(
		actual := success,
		message := "Each callback exception must fail Try"
	).IsFalse();
	Assert.ThatUDInt(
		actual := _Extender.StartCount,
		message := "Start must be observed"
	).ToBe(expected := 1);

	IF _Extender.ThrowAtStart THEN
		Assert.ThatUDInt(
			actual := _Extender.FinishCount,
			message := "Failed start must skip finish"
		).ToBe(expected := 0);
	ELSE
		Assert.ThatUDInt(
			actual := _Extender.FinishCount,
			message := "Finish failure must be observed"
		).ToBe(expected := 1);
	END_IF

	_Extender.Reset();
	success := _Serializer.TrySerialize(
		sourceStructure := _Source,
		extender := _Extender,
		targetJson := _Json,
		jsonSize => jsonSize
	);
	Assert.ThatBool(
		actual := success,
		message := "Writer must be reusable after either callback failure"
	).IsTrue();
	Assert.That(
		actual := _Json,
		message := "Reuse must discard the previous partial document"
	).ToBe(expected := expectedJson);
END_FOR
END_METHOD

(*!
<summary>Restores the fixture before the runner publishes the result.</summary>
<description>
Also runs after an unexpected exception interrupts the case.
</description>
*)
METHOD PROTECTED AfterTest
_Extender.Reset();
END_METHOD

//! <summary>Borrows the concrete class name. Callers must not modify it.</summary>
{attribute 'monitoring' := 'call'}
PROPERTY ClassName : REFERENCE TO STRING
GET
ClassName REF= _ClassName;
END_GET
END_PROPERTY

//! <summary>Borrows the compiler-initialized namespace name. Callers must not modify it.</summary>
{attribute 'monitoring' := 'call'}
PROPERTY NamespaceName : REFERENCE TO STRING
GET
NamespaceName REF= CurrentNamespace.Name;
END_GET
END_PROPERTY

//! <summary>Reports the concrete instance size in bytes.</summary>
{attribute 'monitoring' := 'call'}
PROPERTY SelfSize : ULINT
GET
SelfSize := XSIZEOF(THIS^);
END_GET
END_PROPERTY

END_FUNCTION_BLOCK

// ---- Tests/JSON/AutomaticJsonThrowingCallbackPropagationTest.TcPOU
(*
SPDX-FileCopyrightText: c 2026 Oleksandr Tiutyk <trofimich@gmail.com>
SPDX-License-Identifier: MIT
License: https://opensource.org/license/mit
*)

(*!
<summary>Checks that throwing Create APIs propagate callback failures with their category.</summary>
<description>
Owns persistent native serializer state and any payload buffers used by this case.
Run from one task at a stable address. The caller provides task-boundary exception cleanup.
</description>
*)

{attribute 'no_assign'}
{attribute 'no_explicit_call' := 'do not call this function block directly'}
FUNCTION_BLOCK AutomaticJsonThrowingCallbackPropagationTest EXTENDS TOF_Testing.SingleCycleTest
VAR_STAT
	{attribute 'hide'}
	_ClassName : STRING := __POUNAME();
END_VAR
VAR
	_Serializer : TOF_JSON.AutomaticJsonSerializer;
	_Extender : JsonExtenderProbe;
	_Source : JSON_TEST_VALUE;
	_Json : TOF_Core.JSON_DOCUMENT;
END_VAR

(*!
<summary>Checks that throwing Create APIs propagate callback failures with their category.</summary>
*)
METHOD PROTECTED ExecuteTest
VAR
	exceptionCode : __SYSTEM.ExceptionCode;
	caughtException : TOF_Core.IException;
	standard : TOF_Core.IStandardException;
	sourceInfo : __SYSTEM.VAR_INFO;
	jsonSize : UDINT;
	i : INT;
	scenario : WSTRING(255);
END_VAR
_Source.Number := 42;
_Source.Ready := TRUE;

_Json := '';

_Extender.Reset();

sourceInfo := __VARINFO(_Source);

FOR i := 0 TO 3 DO
	_Extender.Reset();
	_Extender.ThrowAtStart := (i MOD 2) = 0;
	_Extender.ThrowAtFinish := NOT _Extender.ThrowAtStart;
	scenario := TOF_Core.WideStrings.Concat255("Throwing callback case ", TO_WSTRING(i + 1));
	caughtException := 0;
	standard := 0;

	__TRY
		IF i < 2 THEN
			_Serializer.Serialize(
				sourceStructure := _Source,
				extender := _Extender,
				targetJson := _Json,
				jsonSize => jsonSize
			);
		ELSE
			_Serializer.SerializeByVarInfo(
				sourceStructureVarInfo := sourceInfo,
				sourceStructureAddress := ADR(_Source),
				extender := _Extender,
				targetJson := _Json,
				jsonSize => jsonSize
			);
		END_IF
	__CATCH(exceptionCode)
		caughtException := TOF_Core.ExceptionManager.GetLastException(
			exceptionCode := exceptionCode,
			catchPointNamespaceName := CurrentNamespace.Name,
			catchPointPOUName := __POUNAME(),
			catchPointPosition := __POSITION()
		);
	__ENDTRY

	Assert.ThatBool(
		actual := __QUERYINTERFACE(caughtException, standard),
		message := TOF_Core.WideStrings.Concat255(scenario, " must propagate a StandardException")
	).IsTrue();

	IF standard <> 0 THEN
		Assert.ThatWideString(
			actual := standard.SourceMessage,
			message := TOF_Core.WideStrings.Concat255(scenario, " must preserve the injected diagnostic")
		).ToBe(expected := "JSON extender injected failure");
	END_IF
END_FOR
END_METHOD

(*!
<summary>Restores the fixture before the runner publishes the result.</summary>
<description>
Also runs after an unexpected exception interrupts the case.
</description>
*)
METHOD PROTECTED AfterTest
_Extender.Reset();
END_METHOD

//! <summary>Borrows the concrete class name. Callers must not modify it.</summary>
{attribute 'monitoring' := 'call'}
PROPERTY ClassName : REFERENCE TO STRING
GET
ClassName REF= _ClassName;
END_GET
END_PROPERTY

//! <summary>Borrows the compiler-initialized namespace name. Callers must not modify it.</summary>
{attribute 'monitoring' := 'call'}
PROPERTY NamespaceName : REFERENCE TO STRING
GET
NamespaceName REF= CurrentNamespace.Name;
END_GET
END_PROPERTY

//! <summary>Reports the concrete instance size in bytes.</summary>
{attribute 'monitoring' := 'call'}
PROPERTY SelfSize : ULINT
GET
SelfSize := XSIZEOF(THIS^);
END_GET
END_PROPERTY

END_FUNCTION_BLOCK

// ---- Tests/JSON/AutomaticJsonCapacityOverflowAndReuseTest.TcPOU
(*
SPDX-FileCopyrightText: c 2026 Oleksandr Tiutyk <trofimich@gmail.com>
SPDX-License-Identifier: MIT
License: https://opensource.org/license/mit
*)

(*!
<summary>Checks the full 25000-byte text boundary, overflow refusal and subsequent reset.</summary>
<description>
Owns persistent native serializer state and any payload buffers used by this case.
Run from one task at a stable address. The caller provides task-boundary exception cleanup.
</description>
*)

{attribute 'no_assign'}
{attribute 'no_explicit_call' := 'do not call this function block directly'}
FUNCTION_BLOCK AutomaticJsonCapacityOverflowAndReuseTest EXTENDS TOF_Testing.SingleCycleTest
VAR_STAT
	{attribute 'hide'}
	_ClassName : STRING := __POUNAME();
END_VAR
VAR
	_Serializer : TOF_JSON.AutomaticJsonSerializer;
	_Source : JSON_TEST_VALUE;
	_LargeSource : JSON_TEST_LARGE_VALUE;
	_Json : TOF_Core.JSON_DOCUMENT;
END_VAR

(*!
<summary>Checks the full 25000-byte text boundary, overflow refusal and subsequent reset.</summary>
*)
METHOD PROTECTED ExecuteTest
VAR
	caught : BOOL;
	exceptionCode : __SYSTEM.ExceptionCode;
	caughtException : TOF_Core.IException;
	standard : TOF_Core.IStandardException;
	jsonSize : UDINT;
	success : BOOL;
	payloadLength : DINT;
	i : DINT;
	expectedJson : STRING(40) := '{"Number":42,"Ready":true}';
END_VAR
_Source.Number := 42;
_Source.Ready := TRUE;

_Json := '';

_LargeSource.Text := '';
_LargeSource.Marker := 7;

success := _Serializer.TrySerialize(
	sourceStructure := _LargeSource,
	extender := 0,
	targetJson := _Json,
	jsonSize => jsonSize
);
Assert.ThatBool(
	actual := success,
	message := "Empty large structure must serialize"
).IsTrue();

Assert.ThatBool(
	actual := jsonSize > 1 AND_THEN jsonSize < TO_UDINT(SIZEOF(_Json)),
	message := "Reported baseline byte count must allow an exact-capacity payload"
).IsTrue();

IF NOT success OR_ELSE jsonSize <= 1 OR_ELSE jsonSize >= TO_UDINT(SIZEOF(_Json)) THEN
	RETURN;
END_IF

payloadLength := TO_DINT(TO_UDINT(SIZEOF(_Json)) - jsonSize);

IF payloadLength + 1 >= TO_DINT(SIZEOF(_LargeSource.Text)) THEN
	RecordFailure(message := "The boundary fixture must hold the overflow byte and terminator");

	RETURN;
END_IF

// SA0175: Fill an exact ASCII byte count before testing the capacity boundary.
{analysis -175}
FOR i := 0 TO payloadLength - 1 DO
	_LargeSource.Text[i] := BYTE#16#61;
END_FOR

_LargeSource.Text[payloadLength] := BYTE#0;
{analysis +175}

success := _Serializer.TrySerialize(
	sourceStructure := _LargeSource,
	extender := 0,
	targetJson := _Json,
	jsonSize => jsonSize
);
Assert.ThatBool(
	actual := success,
	message := "Exact-capacity document must fit with its terminator"
).IsTrue();
Assert.ThatUDInt(
	actual := jsonSize,
	message := "Exact-capacity copy must include all 25001 bytes"
).ToBe(expected := UDINT#25001);

// SA0175: Inspect the final byte of the destination buffer at the exact-capacity boundary.
{analysis -175}
Assert.ThatByte(
	actual := _Json[TO_DINT(SIZEOF(_Json)) - 1],
	message := "The exact-capacity output must end with a terminator"
).ToBe(expected := BYTE#0);
{analysis +175}

// SA0175: Append exactly one ASCII byte and its terminator within the large source buffer.
{analysis -175}
_LargeSource.Text[payloadLength] := BYTE#16#61;
_LargeSource.Text[payloadLength + 1] := BYTE#0;
{analysis +175}
success := _Serializer.TrySerialize(
	sourceStructure := _LargeSource,
	extender := 0,
	targetJson := _Json,
	jsonSize => jsonSize
);
Assert.ThatBool(
	actual := success,
	message := "One byte beyond capacity must fail Try"
).IsFalse();

__TRY
	_Serializer.Serialize(
		sourceStructure := _LargeSource,
		extender := 0,
		targetJson := _Json,
		jsonSize => jsonSize
	);
__CATCH(exceptionCode)
	caught := TRUE;
	caughtException := TOF_Core.ExceptionManager.GetLastException(
		exceptionCode := exceptionCode,
		catchPointNamespaceName := CurrentNamespace.Name,
		catchPointPOUName := __POUNAME(),
		catchPointPosition := __POSITION()
	);
	Assert.ThatBool(
		actual := __QUERYINTERFACE(caughtException, standard),
		message := "Overflow must report StandardException"
	).IsTrue();
__ENDTRY

Assert.ThatBool(
	actual := caught,
	message := "Throwing Create must reject overflow"
).IsTrue();

success := _Serializer.TrySerialize(
	sourceStructure := _Source,
	extender := 0,
	targetJson := _Json,
	jsonSize => jsonSize
);
Assert.ThatBool(
	actual := success,
	message := "A small document must succeed after overflow"
).IsTrue();
Assert.That(
	actual := _Json,
	message := "Overflow reuse must contain only the new document"
).ToBe(expected := expectedJson);
END_METHOD

//! <summary>Borrows the concrete class name. Callers must not modify it.</summary>
{attribute 'monitoring' := 'call'}
PROPERTY ClassName : REFERENCE TO STRING
GET
ClassName REF= _ClassName;
END_GET
END_PROPERTY

//! <summary>Borrows the compiler-initialized namespace name. Callers must not modify it.</summary>
{attribute 'monitoring' := 'call'}
PROPERTY NamespaceName : REFERENCE TO STRING
GET
NamespaceName REF= CurrentNamespace.Name;
END_GET
END_PROPERTY

//! <summary>Reports the concrete instance size in bytes.</summary>
{attribute 'monitoring' := 'call'}
PROPERTY SelfSize : ULINT
GET
SelfSize := XSIZEOF(THIS^);
END_GET
END_PROPERTY

END_FUNCTION_BLOCK

// ---- Tests/JSON/AutomaticJsonLongUtf8RoundTripTest.TcPOU
(*
SPDX-FileCopyrightText: c 2026 Oleksandr Tiutyk <trofimich@gmail.com>
SPDX-License-Identifier: MIT
License: https://opensource.org/license/mit
*)

(*!
<summary>Checks long UTF-8 text and escaped characters by independent byte comparison.</summary>
<description>
Owns persistent native serializer state and any payload buffers used by this case.
Run from one task at a stable address. The caller provides task-boundary exception cleanup.
</description>
*)

{attribute 'no_assign'}
{attribute 'no_explicit_call' := 'do not call this function block directly'}
FUNCTION_BLOCK AutomaticJsonLongUtf8RoundTripTest EXTENDS TOF_Testing.SingleCycleTest
VAR_STAT
	{attribute 'hide'}
	_ClassName : STRING := __POUNAME();
END_VAR
VAR
	_Serializer : TOF_JSON.AutomaticJsonSerializer;
	_LargeSource : JSON_TEST_LARGE_VALUE;
	_LargeTarget : JSON_TEST_LARGE_VALUE;
	_Json : TOF_Core.JSON_DOCUMENT;
END_VAR

(*!
<summary>Checks long UTF-8 text and escaped characters by independent byte comparison.</summary>
*)
METHOD PROTECTED ExecuteTest
VAR
	i : DINT;
	success : BOOL;
	jsonSize : UDINT;
END_VAR
_Json := '';

_LargeSource.Text := '';
_LargeSource.Marker := 7;
_LargeTarget.Text := '';
_LargeTarget.Marker := 0;

// SA0175: Seed the destination terminator and fill the source with exact UTF-8 and escape bytes.
{analysis -175}
_LargeTarget.Text[305] := BYTE#16#58;

FOR i := 0 TO 299 DO
	_LargeSource.Text[i] := BYTE#16#61;
END_FOR

// UTF-8 U+00E9 followed by quote, backslash, newline and the terminator.
_LargeSource.Text[300] := BYTE#16#C3;
_LargeSource.Text[301] := BYTE#16#A9;
_LargeSource.Text[302] := BYTE#16#22;
_LargeSource.Text[303] := BYTE#16#5C;
_LargeSource.Text[304] := BYTE#16#0A;
_LargeSource.Text[305] := BYTE#0;
{analysis +175}

success := _Serializer.TrySerialize(
	sourceStructure := _LargeSource,
	extender := 0,
	targetJson := _Json,
	jsonSize => jsonSize
);
Assert.ThatBool(
	actual := success,
	message := "Long UTF-8 text must serialize"
).IsTrue();

success := _Serializer.TryDeserialize(json := _Json, targetStructure := _LargeTarget);
Assert.ThatBool(
	actual := success,
	message := "Long UTF-8 text must deserialize"
).IsTrue();

// SA0175: The oracle compares all payload bytes and the terminator, not Unicode character positions.
{analysis -175}
FOR i := 0 TO 305 DO
	Assert.ThatByte(
		actual := _LargeTarget.Text[i],
		message := TOF_Core.WideStrings.Concat255("UTF-8 byte at offset ", TO_WSTRING(i))
	).ToBe(expected := _LargeSource.Text[i]);
END_FOR
{analysis +175}

Assert.ThatDInt(
	actual := _LargeTarget.Marker,
	message := "Long text must preserve the adjacent field"
).ToBe(expected := 7);
END_METHOD

//! <summary>Borrows the concrete class name. Callers must not modify it.</summary>
{attribute 'monitoring' := 'call'}
PROPERTY ClassName : REFERENCE TO STRING
GET
ClassName REF= _ClassName;
END_GET
END_PROPERTY

//! <summary>Borrows the compiler-initialized namespace name. Callers must not modify it.</summary>
{attribute 'monitoring' := 'call'}
PROPERTY NamespaceName : REFERENCE TO STRING
GET
NamespaceName REF= CurrentNamespace.Name;
END_GET
END_PROPERTY

//! <summary>Reports the concrete instance size in bytes.</summary>
{attribute 'monitoring' := 'call'}
PROPERTY SelfSize : ULINT
GET
SelfSize := XSIZEOF(THIS^);
END_GET
END_PROPERTY

END_FUNCTION_BLOCK

// ---- Tests/JSON/AutomaticJsonDecimalPlacesReadbackTest.TcPOU
(*
SPDX-FileCopyrightText: c 2026 Oleksandr Tiutyk <trofimich@gmail.com>
SPDX-License-Identifier: MIT
License: https://opensource.org/license/mit
*)

(*!
<summary>Checks native decimal-place configuration and readback without inventing a clamp policy.</summary>
<description>
Owns persistent native serializer state and any payload buffers used by this case.
Run from one task at a stable address. The caller provides task-boundary exception cleanup.
</description>
*)

{attribute 'no_assign'}
{attribute 'no_explicit_call' := 'do not call this function block directly'}
FUNCTION_BLOCK AutomaticJsonDecimalPlacesReadbackTest EXTENDS TOF_Testing.SingleCycleTest
VAR_STAT
	{attribute 'hide'}
	_ClassName : STRING := __POUNAME();
END_VAR
VAR
	_Serializer : TOF_JSON.AutomaticJsonSerializer;
END_VAR

(*!
<summary>Checks native decimal-place configuration and readback without inventing a clamp policy.</summary>
*)
METHOD PROTECTED ExecuteTest
_Serializer.DecimalPlaces := 3;
Assert.ThatDInt(
	actual := _Serializer.DecimalPlaces,
	message := "Native decimal setting must be readable"
).ToBe(expected := 3);

_Serializer.DecimalPlaces := 6;

Assert.ThatDInt(
	actual := _Serializer.DecimalPlaces,
	message := "A later native decimal setting must replace the first"
).ToBe(expected := DINT#6);
END_METHOD

//! <summary>Borrows the concrete class name. Callers must not modify it.</summary>
{attribute 'monitoring' := 'call'}
PROPERTY ClassName : REFERENCE TO STRING
GET
ClassName REF= _ClassName;
END_GET
END_PROPERTY

//! <summary>Borrows the compiler-initialized namespace name. Callers must not modify it.</summary>
{attribute 'monitoring' := 'call'}
PROPERTY NamespaceName : REFERENCE TO STRING
GET
NamespaceName REF= CurrentNamespace.Name;
END_GET
END_PROPERTY

//! <summary>Reports the concrete instance size in bytes.</summary>
{attribute 'monitoring' := 'call'}
PROPERTY SelfSize : ULINT
GET
SelfSize := XSIZEOF(THIS^);
END_GET
END_PROPERTY

END_FUNCTION_BLOCK

// ---- Tests/Collections/Static/StaticQueueTestGroup.TcPOU
(*
SPDX-FileCopyrightText: c 2026 Oleksandr Tiutyk <trofimich@gmail.com>
SPDX-License-Identifier: MIT
License: https://opensource.org/license/mit
*)

(*!
<summary>Groups fixed-capacity queue lookup, FIFO, clear and overflow cases.</summary>
<description>
Owns the independent child instances and their fixed registration array. Use from one PLC task at a stable address.
</description>
*)

{attribute 'no_assign'}
{attribute 'no_explicit_call' := 'do not call this function block directly'}
FUNCTION_BLOCK StaticQueueTestGroup EXTENDS TOF_Testing.TestGroup<6>
VAR_STAT
	{attribute 'hide'}
	_ClassName : STRING := __POUNAME();
END_VAR
VAR
	_Contains : StaticQueueContainsTest(name := "Contains", parent := THIS^);
	_ContainsGeneric : StaticQueueContainsGenericTest(name := "ContainsGeneric", parent := THIS^);
	_EnqueueAndPeek : StaticQueueEnqueueAndPeekTest(name := "EnqueueAndPeek", parent := THIS^);
	_Clear : StaticQueueClearTest(name := "Clear", parent := THIS^);
	_RemoveFirst : StaticQueueRemoveFirstTest(name := "RemoveFirst", parent := THIS^);
	_Overflow : StaticQueueOverflowTest(name := "Overflow", parent := THIS^);

	_Children : ARRAY [0.._ChildCount - 1] OF TOF_Testing.ITestElement :=
	[
		_Contains,
		_ContainsGeneric,
		_EnqueueAndPeek,
		_Clear,
		_RemoveFirst,
		_Overflow
	];
END_VAR

//! <summary>Borrows the fixed child array. Callers must not modify it.</summary>
{attribute 'monitoring' := 'call'}
PROPERTY Children : REFERENCE TO ARRAY [0.._ChildCount - 1] OF TOF_Testing.ITestElement
GET
Children REF= _Children;
END_GET
END_PROPERTY

//! <summary>Borrows the concrete class name. Callers must not modify it.</summary>
{attribute 'monitoring' := 'call'}
PROPERTY ClassName : REFERENCE TO STRING
GET
ClassName REF= _ClassName;
END_GET
END_PROPERTY

//! <summary>Borrows the compiler-initialized namespace name. Callers must not modify it.</summary>
{attribute 'monitoring' := 'call'}
PROPERTY NamespaceName : REFERENCE TO STRING
GET
NamespaceName REF= CurrentNamespace.Name;
END_GET
END_PROPERTY

//! <summary>Reports the concrete instance size in bytes.</summary>
{attribute 'monitoring' := 'call'}
PROPERTY SelfSize : ULINT
GET
SelfSize := XSIZEOF(THIS^);
END_GET
END_PROPERTY

END_FUNCTION_BLOCK

// ---- Tests/Collections/Static/StaticQueueContainsTest.TcPOU
(*
SPDX-FileCopyrightText: c 2026 Oleksandr Tiutyk <trofimich@gmail.com>
SPDX-License-Identifier: MIT
License: https://opensource.org/license/mit
*)

(*!
<summary>Checks ANY lookup of present and absent values without changing the queue.</summary>
<description>
Owns an inline queue and its copied entry payloads. Run from one task at a stable address.
Teardown clears surviving entries before publication, including after an aborted case.
</description>
*)

{attribute 'no_assign'}
{attribute 'no_explicit_call' := 'do not call this function block directly'}
FUNCTION_BLOCK StaticQueueContainsTest EXTENDS TOF_Testing.SingleCycleTest
VAR_STAT
	{attribute 'hide'}
	_ClassName : STRING := __POUNAME();
END_VAR
VAR
	_Queue : TOF_Collections.Queue<3>(valueValidator := 0);
END_VAR

(*!
<summary>Checks ANY lookup of present and absent values without changing the queue.</summary>
*)
METHOD PROTECTED ExecuteTest
VAR
	values : ARRAY [1..4] OF INT := [11, 22, 33, 44];
END_VAR
Assert.ThatBool(
	actual := _Queue.Contains(value := values[1]),
	message := "An empty queue must report absence"
).IsFalse();

_Queue
	.EnqueueCopy(value := values[1])
	.EnqueueCopy(value := values[2])
	.EnqueueCopy(value := values[3]);

Assert.ThatBool(
	actual := _Queue.Contains(value := values[1]),
	message := "Contains must find the head"
).IsTrue();

Assert.ThatBool(
	actual := _Queue.Contains(value := values[3]),
	message := "Contains must find the tail"
).IsTrue();

Assert.ThatBool(
	actual := _Queue.Contains(value := values[4]),
	message := "Contains must report a missing value"
).IsFalse();

Assert.ThatDInt(
	actual := _Queue.Length,
	message := "Lookup must preserve all three entries"
).ToBe(expected := DINT#3);

Assert.ThatInt(
	actual := _Queue.Peek().AsInt(),
	message := "Lookup must preserve the head"
).ToBe(expected := values[1]);
END_METHOD

(*!
<summary>Restores the fixture before the runner publishes the result.</summary>
<description>
Also runs after an unexpected exception interrupts the case.
</description>
*)
METHOD PROTECTED AfterTest
_Queue.Clear();
END_METHOD

//! <summary>Borrows the concrete class name. Callers must not modify it.</summary>
{attribute 'monitoring' := 'call'}
PROPERTY ClassName : REFERENCE TO STRING
GET
ClassName REF= _ClassName;
END_GET
END_PROPERTY

//! <summary>Borrows the compiler-initialized namespace name. Callers must not modify it.</summary>
{attribute 'monitoring' := 'call'}
PROPERTY NamespaceName : REFERENCE TO STRING
GET
NamespaceName REF= CurrentNamespace.Name;
END_GET
END_PROPERTY

//! <summary>Reports the concrete instance size in bytes.</summary>
{attribute 'monitoring' := 'call'}
PROPERTY SelfSize : ULINT
GET
SelfSize := XSIZEOF(THIS^);
END_GET
END_PROPERTY

END_FUNCTION_BLOCK

// ---- Tests/Collections/Static/StaticQueueContainsGenericTest.TcPOU
(*
SPDX-FileCopyrightText: c 2026 Oleksandr Tiutyk <trofimich@gmail.com>
SPDX-License-Identifier: MIT
License: https://opensource.org/license/mit
*)

(*!
<summary>Checks generic lookup with independent borrowed query values.</summary>
<description>
Owns an inline queue and its copied entry payloads. Run from one task at a stable address.
Teardown clears surviving entries before publication, including after an aborted case.
</description>
*)

{attribute 'no_assign'}
{attribute 'no_explicit_call' := 'do not call this function block directly'}
FUNCTION_BLOCK StaticQueueContainsGenericTest EXTENDS TOF_Testing.SingleCycleTest
VAR_STAT
	{attribute 'hide'}
	_ClassName : STRING := __POUNAME();
END_VAR
VAR
	_Queue : TOF_Collections.Queue<3>(valueValidator := 0);
END_VAR

(*!
<summary>Checks generic lookup with independent borrowed query values.</summary>
*)
METHOD PROTECTED ExecuteTest
VAR
	values : ARRAY [1..4] OF INT := [11, 22, 33, 44];
	query : TOF_Core.GENERIC_VALUE;
END_VAR
_Queue
	.EnqueueCopy(value := values[1])
	.EnqueueCopy(value := values[2])
	.EnqueueCopy(value := values[3]);

query := TOF_Core.GenericValueFactory.FromIntReference(value := values[1]);
Assert.ThatBool(
	actual := _Queue.ContainsGeneric(value := query, releaseValue := FALSE),
	message := "Generic lookup must find the head"
).IsTrue();

query := TOF_Core.GenericValueFactory.FromIntReference(value := values[3]);
Assert.ThatBool(
	actual := _Queue.ContainsGeneric(value := query, releaseValue := FALSE),
	message := "Generic lookup must find the tail"
).IsTrue();

query := TOF_Core.GenericValueFactory.FromIntReference(value := values[4]);
Assert.ThatBool(
	actual := _Queue.ContainsGeneric(value := query, releaseValue := FALSE),
	message := "Generic lookup must report a missing value"
).IsFalse();

Assert.ThatDInt(
	actual := _Queue.Length,
	message := "Generic lookup must preserve queue length"
).ToBe(expected := DINT#3);
END_METHOD

(*!
<summary>Restores the fixture before the runner publishes the result.</summary>
<description>
Also runs after an unexpected exception interrupts the case.
</description>
*)
METHOD PROTECTED AfterTest
_Queue.Clear();
END_METHOD

//! <summary>Borrows the concrete class name. Callers must not modify it.</summary>
{attribute 'monitoring' := 'call'}
PROPERTY ClassName : REFERENCE TO STRING
GET
ClassName REF= _ClassName;
END_GET
END_PROPERTY

//! <summary>Borrows the compiler-initialized namespace name. Callers must not modify it.</summary>
{attribute 'monitoring' := 'call'}
PROPERTY NamespaceName : REFERENCE TO STRING
GET
NamespaceName REF= CurrentNamespace.Name;
END_GET
END_PROPERTY

//! <summary>Reports the concrete instance size in bytes.</summary>
{attribute 'monitoring' := 'call'}
PROPERTY SelfSize : ULINT
GET
SelfSize := XSIZEOF(THIS^);
END_GET
END_PROPERTY

END_FUNCTION_BLOCK

// ---- Tests/Collections/Static/StaticQueueEnqueueAndPeekTest.TcPOU
(*
SPDX-FileCopyrightText: c 2026 Oleksandr Tiutyk <trofimich@gmail.com>
SPDX-License-Identifier: MIT
License: https://opensource.org/license/mit
*)

(*!
<summary>Checks FIFO head, length and copy independence during enqueue.</summary>
<description>
Owns an inline queue and its copied entry payloads. Run from one task at a stable address.
Teardown clears surviving entries before publication, including after an aborted case.
</description>
*)

{attribute 'no_assign'}
{attribute 'no_explicit_call' := 'do not call this function block directly'}
FUNCTION_BLOCK StaticQueueEnqueueAndPeekTest EXTENDS TOF_Testing.SingleCycleTest
VAR_STAT
	{attribute 'hide'}
	_ClassName : STRING := __POUNAME();
END_VAR
VAR
	_Queue : TOF_Collections.Queue<3>(valueValidator := 0);
END_VAR

(*!
<summary>Checks FIFO head, length and copy independence during enqueue.</summary>
*)
METHOD PROTECTED ExecuteTest
VAR
	values : ARRAY [1..4] OF INT := [11, 22, 33, 44];
END_VAR
_Queue.EnqueueCopy(value := values[1]);
values[1] := 111;

Assert.ThatInt(
	actual := _Queue.Peek().AsInt(),
	message := "Changing the source must preserve the copied head"
).ToBe(expected := INT#11);

_Queue.EnqueueCopy(value := values[2]);

Assert.ThatInt(
	actual := _Queue.Peek().AsInt(),
	message := "Enqueueing the second entry must preserve the head"
).ToBe(expected := INT#11);

_Queue.EnqueueCopy(value := values[3]);

Assert.ThatInt(
	actual := _Queue.Peek().AsInt(),
	message := "Enqueueing the third entry must preserve the head"
).ToBe(expected := INT#11);

Assert.ThatBool(
	actual := _Queue.Full AND_THEN _Queue.Length = 3,
	message := "Only enqueue must advance length while peeking leaves the queue full"
).IsTrue();
END_METHOD

(*!
<summary>Restores the fixture before the runner publishes the result.</summary>
<description>
Also runs after an unexpected exception interrupts the case.
</description>
*)
METHOD PROTECTED AfterTest
_Queue.Clear();
END_METHOD

//! <summary>Borrows the concrete class name. Callers must not modify it.</summary>
{attribute 'monitoring' := 'call'}
PROPERTY ClassName : REFERENCE TO STRING
GET
ClassName REF= _ClassName;
END_GET
END_PROPERTY

//! <summary>Borrows the compiler-initialized namespace name. Callers must not modify it.</summary>
{attribute 'monitoring' := 'call'}
PROPERTY NamespaceName : REFERENCE TO STRING
GET
NamespaceName REF= CurrentNamespace.Name;
END_GET
END_PROPERTY

//! <summary>Reports the concrete instance size in bytes.</summary>
{attribute 'monitoring' := 'call'}
PROPERTY SelfSize : ULINT
GET
SelfSize := XSIZEOF(THIS^);
END_GET
END_PROPERTY

END_FUNCTION_BLOCK

// ---- Tests/Collections/Static/StaticQueueClearTest.TcPOU
(*
SPDX-FileCopyrightText: c 2026 Oleksandr Tiutyk <trofimich@gmail.com>
SPDX-License-Identifier: MIT
License: https://opensource.org/license/mit
*)

(*!
<summary>Checks populated clear, retained capacity and reuse.</summary>
<description>
Owns an inline queue and its copied entry payloads. Run from one task at a stable address.
Teardown clears surviving entries before publication, including after an aborted case.
</description>
*)

{attribute 'no_assign'}
{attribute 'no_explicit_call' := 'do not call this function block directly'}
FUNCTION_BLOCK StaticQueueClearTest EXTENDS TOF_Testing.SingleCycleTest
VAR_STAT
	{attribute 'hide'}
	_ClassName : STRING := __POUNAME();
END_VAR
VAR
	_Queue : TOF_Collections.Queue<3>(valueValidator := 0);
END_VAR

(*!
<summary>Checks populated clear, retained capacity and reuse.</summary>
*)
METHOD PROTECTED ExecuteTest
VAR
	values : ARRAY [1..4] OF INT := [11, 22, 33, 44];
END_VAR
_Queue
	.EnqueueCopy(value := values[1])
	.EnqueueCopy(value := values[2])
	.EnqueueCopy(value := values[3]);

Assert.ThatBool(
	actual := _Queue.Full AND_THEN _Queue.Length = 3,
	message := "The clear fixture must start full"
).IsTrue();

_Queue.Clear();

Assert.ThatBool(
	actual := _Queue.Empty AND_THEN _Queue.Length = 0 AND_THEN NOT _Queue.Full,
	message := "Clearing a populated queue must remove all entries"
).IsTrue();

Assert.ThatDInt(
	actual := _Queue.Capacity,
	message := "Clearing must preserve inline capacity"
).ToBe(expected := DINT#3);

Assert.ThatBool(
	actual := _Queue.Contains(value := values[3]),
	message := "Clearing must hide the previous tail"
).IsFalse();

_Queue.Clear();
_Queue.EnqueueCopy(value := values[4]);

Assert.ThatInt(
	actual := _Queue.Peek().AsInt(),
	message := "The cleared queue must accept a fresh head"
).ToBe(expected := values[4]);

Assert.ThatDInt(
	actual := _Queue.Length,
	message := "Reuse must leave only the fresh entry"
).ToBe(expected := DINT#1);
END_METHOD

(*!
<summary>Restores the fixture before the runner publishes the result.</summary>
<description>
Also runs after an unexpected exception interrupts the case.
</description>
*)
METHOD PROTECTED AfterTest
_Queue.Clear();
END_METHOD

//! <summary>Borrows the concrete class name. Callers must not modify it.</summary>
{attribute 'monitoring' := 'call'}
PROPERTY ClassName : REFERENCE TO STRING
GET
ClassName REF= _ClassName;
END_GET
END_PROPERTY

//! <summary>Borrows the compiler-initialized namespace name. Callers must not modify it.</summary>
{attribute 'monitoring' := 'call'}
PROPERTY NamespaceName : REFERENCE TO STRING
GET
NamespaceName REF= CurrentNamespace.Name;
END_GET
END_PROPERTY

//! <summary>Reports the concrete instance size in bytes.</summary>
{attribute 'monitoring' := 'call'}
PROPERTY SelfSize : ULINT
GET
SelfSize := XSIZEOF(THIS^);
END_GET
END_PROPERTY

END_FUNCTION_BLOCK

// ---- Tests/Collections/Static/StaticQueueRemoveFirstTest.TcPOU
(*
SPDX-FileCopyrightText: c 2026 Oleksandr Tiutyk <trofimich@gmail.com>
SPDX-License-Identifier: MIT
License: https://opensource.org/license/mit
*)

(*!
<summary>Checks FIFO removal through empty and reuse after a rejected removal.</summary>
<description>
Owns an inline queue and its copied entry payloads. Run from one task at a stable address.
Teardown clears surviving entries before publication, including after an aborted case.
</description>
*)

{attribute 'no_assign'}
{attribute 'no_explicit_call' := 'do not call this function block directly'}
FUNCTION_BLOCK StaticQueueRemoveFirstTest EXTENDS TOF_Testing.SingleCycleTest
VAR_STAT
	{attribute 'hide'}
	_ClassName : STRING := __POUNAME();
END_VAR
VAR
	_Queue : TOF_Collections.Queue<3>(valueValidator := 0);
END_VAR

(*!
<summary>Checks FIFO removal through empty and reuse after a rejected removal.</summary>
*)
METHOD PROTECTED ExecuteTest
VAR
	values : ARRAY [1..4] OF INT := [11, 22, 33, 44];

	exceptionCode : __SYSTEM.ExceptionCode;
	caught : TOF_Core.IException;
	emptyException : TOF_Core.ICollectionEmptyException;
END_VAR
_Queue
	.EnqueueCopy(value := values[1])
	.EnqueueCopy(value := values[2])
	.EnqueueCopy(value := values[3]);

_Queue.RemoveFirst();

Assert.ThatInt(
	actual := _Queue.Peek().AsInt(),
	message := "The second entry must become the head after the first removal"
).ToBe(expected := values[2]);

Assert.ThatDInt(
	actual := _Queue.Length,
	message := "Removing the first entry must leave two entries"
).ToBe(expected := DINT#2);

_Queue.RemoveFirst();

Assert.ThatInt(
	actual := _Queue.Peek().AsInt(),
	message := "The third entry must become the head after the second removal"
).ToBe(expected := values[3]);

_Queue.RemoveFirst();

Assert.ThatBool(
	actual := _Queue.Empty,
	message := "Removing the final entry must leave an empty queue"
).IsTrue();

__TRY
	_Queue.RemoveFirst();
__CATCH(exceptionCode)
	caught := TOF_Core.ExceptionManager.GetLastException(
		exceptionCode := exceptionCode,
		catchPointNamespaceName := NamespaceName,
		catchPointPOUName := __POUNAME(),
		catchPointPosition := __POSITION()
	);
__ENDTRY

Assert.ThatBool(
	actual := __QUERYINTERFACE(caught, emptyException),
	message := "Removing from an empty queue must raise CollectionEmptyException"
).IsTrue();

Assert.ThatDInt(
	actual := _Queue.Length,
	message := "Rejected removal must preserve empty length"
).ToBe(expected := DINT#0);

_Queue.EnqueueCopy(value := values[4]);

Assert.ThatInt(
	actual := _Queue.Peek().AsInt(),
	message := "Reuse after rejected removal must expose the new head"
).ToBe(expected := values[4]);
END_METHOD

(*!
<summary>Restores the fixture before the runner publishes the result.</summary>
<description>
Also runs after an unexpected exception interrupts the case.
</description>
*)
METHOD PROTECTED AfterTest
_Queue.Clear();
END_METHOD

//! <summary>Borrows the concrete class name. Callers must not modify it.</summary>
{attribute 'monitoring' := 'call'}
PROPERTY ClassName : REFERENCE TO STRING
GET
ClassName REF= _ClassName;
END_GET
END_PROPERTY

//! <summary>Borrows the compiler-initialized namespace name. Callers must not modify it.</summary>
{attribute 'monitoring' := 'call'}
PROPERTY NamespaceName : REFERENCE TO STRING
GET
NamespaceName REF= CurrentNamespace.Name;
END_GET
END_PROPERTY

//! <summary>Reports the concrete instance size in bytes.</summary>
{attribute 'monitoring' := 'call'}
PROPERTY SelfSize : ULINT
GET
SelfSize := XSIZEOF(THIS^);
END_GET
END_PROPERTY

END_FUNCTION_BLOCK

// ---- Tests/Collections/Static/StaticQueueOverflowTest.TcPOU
(*
SPDX-FileCopyrightText: c 2026 Oleksandr Tiutyk <trofimich@gmail.com>
SPDX-License-Identifier: MIT
License: https://opensource.org/license/mit
*)

(*!
<summary>Checks full-capacity rejection without losing entries or FIFO order.</summary>
<description>
Owns an inline queue and its copied entry payloads. Run from one task at a stable address.
Teardown clears surviving entries before publication, including after an aborted case.
</description>
*)

{attribute 'no_assign'}
{attribute 'no_explicit_call' := 'do not call this function block directly'}
FUNCTION_BLOCK StaticQueueOverflowTest EXTENDS TOF_Testing.SingleCycleTest
VAR_STAT
	{attribute 'hide'}
	_ClassName : STRING := __POUNAME();
END_VAR
VAR
	_Queue : TOF_Collections.Queue<3>(valueValidator := 0);
END_VAR

(*!
<summary>Checks full-capacity rejection without losing entries or FIFO order.</summary>
*)
METHOD PROTECTED ExecuteTest
VAR
	values : ARRAY [1..4] OF INT := [11, 22, 33, 44];
	i : DINT;

	exceptionCode : __SYSTEM.ExceptionCode;
	caught : TOF_Core.IException;
	fullException : TOF_Core.IStaticCollectionFullException;
END_VAR
_Queue
	.EnqueueCopy(value := values[1])
	.EnqueueCopy(value := values[2])
	.EnqueueCopy(value := values[3]);

__TRY
	_Queue.EnqueueCopy(value := values[4]);
__CATCH(exceptionCode)
	caught := TOF_Core.ExceptionManager.GetLastException(
		exceptionCode := exceptionCode,
		catchPointNamespaceName := NamespaceName,
		catchPointPOUName := __POUNAME(),
		catchPointPosition := __POSITION()
	);
__ENDTRY

Assert.ThatBool(
	actual := __QUERYINTERFACE(caught, fullException),
	message := "A full queue must raise StaticCollectionFullException"
).IsTrue();

Assert.ThatBool(
	actual := _Queue.Full AND_THEN _Queue.Length = 3 AND_THEN _Queue.Capacity = 3,
	message := "Rejected enqueue must preserve the full queue and its capacity"
).IsTrue();

FOR i := 1 TO 3 DO
	Assert.ThatInt(
		actual := _Queue.GetByIndex(index := i - 1).AsInt(),
		message := "A rejected enqueue must preserve every entry in FIFO order"
	).ToBe(expected := values[i]);
END_FOR

_Queue.RemoveFirst();
_Queue.EnqueueCopy(value := values[4]);

Assert.ThatBool(
	actual := _Queue.Full,
	message := "Enqueue must succeed after freeing a slot"
).IsTrue();

Assert.ThatInt(
	actual := _Queue.Peek().AsInt(),
	message := "Enqueue after freeing a slot must preserve the current head"
).ToBe(expected := values[2]);

Assert.ThatInt(
	actual := _Queue.GetByIndex(index := 2).AsInt(),
	message := "The new entry must become the tail"
).ToBe(expected := values[4]);
END_METHOD

(*!
<summary>Restores the fixture before the runner publishes the result.</summary>
<description>
Also runs after an unexpected exception interrupts the case.
</description>
*)
METHOD PROTECTED AfterTest
_Queue.Clear();
END_METHOD

//! <summary>Borrows the concrete class name. Callers must not modify it.</summary>
{attribute 'monitoring' := 'call'}
PROPERTY ClassName : REFERENCE TO STRING
GET
ClassName REF= _ClassName;
END_GET
END_PROPERTY

//! <summary>Borrows the compiler-initialized namespace name. Callers must not modify it.</summary>
{attribute 'monitoring' := 'call'}
PROPERTY NamespaceName : REFERENCE TO STRING
GET
NamespaceName REF= CurrentNamespace.Name;
END_GET
END_PROPERTY

//! <summary>Reports the concrete instance size in bytes.</summary>
{attribute 'monitoring' := 'call'}
PROPERTY SelfSize : ULINT
GET
SelfSize := XSIZEOF(THIS^);
END_GET
END_PROPERTY

END_FUNCTION_BLOCK

// ---- Tests/Collections/Dynamic/DynamicQueueTestGroup.TcPOU
(*
SPDX-FileCopyrightText: c 2026 Oleksandr Tiutyk <trofimich@gmail.com>
SPDX-License-Identifier: MIT
License: https://opensource.org/license/mit
*)

(*!
<summary>Groups dynamic queue lookup, FIFO, growth and clear cases.</summary>
<description>
Owns the independent child instances and their fixed registration array. Use from one PLC task at a stable address.
</description>
*)

{attribute 'no_assign'}
{attribute 'no_explicit_call' := 'do not call this function block directly'}
FUNCTION_BLOCK DynamicQueueTestGroup EXTENDS TOF_Testing.TestGroup<5>
VAR_STAT
	{attribute 'hide'}
	_ClassName : STRING := __POUNAME();
END_VAR
VAR
	_Contains : DynamicQueueContainsTest(name := "Contains", parent := THIS^);
	_ContainsGeneric : DynamicQueueContainsGenericTest(name := "ContainsGeneric", parent := THIS^);
	_EnqueueAndPeek : DynamicQueueEnqueueAndPeekTest(name := "EnqueueAndPeek", parent := THIS^);
	_Clear : DynamicQueueClearTest(name := "Clear", parent := THIS^);
	_RemoveFirst : DynamicQueueRemoveFirstTest(name := "RemoveFirst", parent := THIS^);

	_Children : ARRAY [0.._ChildCount - 1] OF TOF_Testing.ITestElement :=
	[
		_Contains,
		_ContainsGeneric,
		_EnqueueAndPeek,
		_Clear,
		_RemoveFirst
	];
END_VAR

//! <summary>Borrows the fixed child array. Callers must not modify it.</summary>
{attribute 'monitoring' := 'call'}
PROPERTY Children : REFERENCE TO ARRAY [0.._ChildCount - 1] OF TOF_Testing.ITestElement
GET
Children REF= _Children;
END_GET
END_PROPERTY

//! <summary>Borrows the concrete class name. Callers must not modify it.</summary>
{attribute 'monitoring' := 'call'}
PROPERTY ClassName : REFERENCE TO STRING
GET
ClassName REF= _ClassName;
END_GET
END_PROPERTY

//! <summary>Borrows the compiler-initialized namespace name. Callers must not modify it.</summary>
{attribute 'monitoring' := 'call'}
PROPERTY NamespaceName : REFERENCE TO STRING
GET
NamespaceName REF= CurrentNamespace.Name;
END_GET
END_PROPERTY

//! <summary>Reports the concrete instance size in bytes.</summary>
{attribute 'monitoring' := 'call'}
PROPERTY SelfSize : ULINT
GET
SelfSize := XSIZEOF(THIS^);
END_GET
END_PROPERTY

END_FUNCTION_BLOCK

// ---- Tests/Collections/Dynamic/DynamicQueueContainsTest.TcPOU
(*
SPDX-FileCopyrightText: c 2026 Oleksandr Tiutyk <trofimich@gmail.com>
SPDX-License-Identifier: MIT
License: https://opensource.org/license/mit
*)

(*!
<summary>Checks ANY lookup after growth and head removal.</summary>
<description>
Owns a dynamic queue and copied payloads at a stable address. Run from one task.
Teardown clears surviving entries and releases dynamic capacity.
</description>
*)

{attribute 'no_assign'}
{attribute 'no_explicit_call' := 'do not call this function block directly'}
FUNCTION_BLOCK DynamicQueueContainsTest EXTENDS TOF_Testing.SingleCycleTest
VAR_STAT
	{attribute 'hide'}
	_ClassName : STRING := __POUNAME();
END_VAR
VAR
	_Queue : TOF_Collections.Queue<0>(valueValidator := 0);
END_VAR

(*!
<summary>Checks ANY lookup after growth and head removal.</summary>
*)
METHOD PROTECTED ExecuteTest
VAR
	values : ARRAY [1..4] OF INT := [11, 22, 33, 44];
END_VAR
_Queue.DefaultDynamicAllocationElementCount := BYTE#2;

_Queue
	.EnqueueCopy(value := values[1])
	.EnqueueCopy(value := values[2])
	.EnqueueCopy(value := values[3]);

Assert.ThatBool(
	actual := _Queue.Contains(value := values[1]),
	message := "Lookup must find the original head after growth"
).IsTrue();

Assert.ThatBool(
	actual := _Queue.Contains(value := values[3]),
	message := "Lookup must find the entry appended during growth"
).IsTrue();

Assert.ThatBool(
	actual := _Queue.Contains(value := values[4]),
	message := "Lookup must reject an absent value"
).IsFalse();

_Queue.RemoveFirst();

Assert.ThatBool(
	actual := _Queue.Contains(value := values[1]),
	message := "Lookup must ignore the removed head"
).IsFalse();

Assert.ThatDInt(
	actual := _Queue.Length,
	message := "Lookup must preserve the two live entries"
).ToBe(expected := DINT#2);

Assert.ThatInt(
	actual := _Queue.Peek().AsInt(),
	message := "Lookup must preserve the current head"
).ToBe(expected := values[2]);
END_METHOD

(*!
<summary>Clears the fixture before the runner publishes the result.</summary>
<description>
Also runs after an unexpected exception interrupts the case.
</description>
*)
METHOD PROTECTED AfterTest
_Queue.Clear();
END_METHOD

//! <summary>Borrows the concrete class name. Callers must not modify it.</summary>
{attribute 'monitoring' := 'call'}
PROPERTY ClassName : REFERENCE TO STRING
GET
ClassName REF= _ClassName;
END_GET
END_PROPERTY

//! <summary>Borrows the compiler-initialized namespace name. Callers must not modify it.</summary>
{attribute 'monitoring' := 'call'}
PROPERTY NamespaceName : REFERENCE TO STRING
GET
NamespaceName REF= CurrentNamespace.Name;
END_GET
END_PROPERTY

//! <summary>Reports the concrete instance size in bytes.</summary>
{attribute 'monitoring' := 'call'}
PROPERTY SelfSize : ULINT
GET
SelfSize := XSIZEOF(THIS^);
END_GET
END_PROPERTY

END_FUNCTION_BLOCK

// ---- Tests/Collections/Dynamic/DynamicQueueContainsGenericTest.TcPOU
(*
SPDX-FileCopyrightText: c 2026 Oleksandr Tiutyk <trofimich@gmail.com>
SPDX-License-Identifier: MIT
License: https://opensource.org/license/mit
*)

(*!
<summary>Checks generic lookup in grown and compacted dynamic storage.</summary>
<description>
Owns a dynamic queue and copied payloads at a stable address. Run from one task.
Teardown clears surviving entries and releases dynamic capacity.
</description>
*)

{attribute 'no_assign'}
{attribute 'no_explicit_call' := 'do not call this function block directly'}
FUNCTION_BLOCK DynamicQueueContainsGenericTest EXTENDS TOF_Testing.SingleCycleTest
VAR_STAT
	{attribute 'hide'}
	_ClassName : STRING := __POUNAME();
END_VAR
VAR
	_Queue : TOF_Collections.Queue<0>(valueValidator := 0);
END_VAR

(*!
<summary>Checks generic lookup in grown and compacted dynamic storage.</summary>
*)
METHOD PROTECTED ExecuteTest
VAR
	values : ARRAY [1..4] OF INT := [11, 22, 33, 44];
	query : TOF_Core.GENERIC_VALUE;
END_VAR
_Queue.DefaultDynamicAllocationElementCount := BYTE#2;

_Queue
	.EnqueueCopy(value := values[1])
	.EnqueueCopy(value := values[2])
	.EnqueueCopy(value := values[3]);

query := TOF_Core.GenericValueFactory.FromIntReference(value := values[1]);
Assert.ThatBool(
	actual := _Queue.ContainsGeneric(value := query, releaseValue := FALSE),
	message := "Generic lookup must find the original head"
).IsTrue();

query := TOF_Core.GenericValueFactory.FromIntReference(value := values[3]);
Assert.ThatBool(
	actual := _Queue.ContainsGeneric(value := query, releaseValue := FALSE),
	message := "Generic lookup must find the new tail"
).IsTrue();

query := TOF_Core.GenericValueFactory.FromIntReference(value := values[4]);
Assert.ThatBool(
	actual := _Queue.ContainsGeneric(value := query, releaseValue := FALSE),
	message := "Generic lookup must reject an absent value"
).IsFalse();

_Queue.RemoveFirst();

query := TOF_Core.GenericValueFactory.FromIntReference(value := values[1]);
Assert.ThatBool(
	actual := _Queue.ContainsGeneric(value := query, releaseValue := FALSE),
	message := "Generic lookup must ignore the removed head"
).IsFalse();

Assert.ThatDInt(
	actual := _Queue.Length,
	message := "Generic lookup must preserve the two live entries"
).ToBe(expected := DINT#2);
END_METHOD

(*!
<summary>Clears the fixture before the runner publishes the result.</summary>
<description>
Also runs after an unexpected exception interrupts the case.
</description>
*)
METHOD PROTECTED AfterTest
_Queue.Clear();
END_METHOD

//! <summary>Borrows the concrete class name. Callers must not modify it.</summary>
{attribute 'monitoring' := 'call'}
PROPERTY ClassName : REFERENCE TO STRING
GET
ClassName REF= _ClassName;
END_GET
END_PROPERTY

//! <summary>Borrows the compiler-initialized namespace name. Callers must not modify it.</summary>
{attribute 'monitoring' := 'call'}
PROPERTY NamespaceName : REFERENCE TO STRING
GET
NamespaceName REF= CurrentNamespace.Name;
END_GET
END_PROPERTY

//! <summary>Reports the concrete instance size in bytes.</summary>
{attribute 'monitoring' := 'call'}
PROPERTY SelfSize : ULINT
GET
SelfSize := XSIZEOF(THIS^);
END_GET
END_PROPERTY

END_FUNCTION_BLOCK

// ---- Tests/Collections/Dynamic/DynamicQueueEnqueueAndPeekTest.TcPOU
(*
SPDX-FileCopyrightText: c 2026 Oleksandr Tiutyk <trofimich@gmail.com>
SPDX-License-Identifier: MIT
License: https://opensource.org/license/mit
*)

(*!
<summary>Checks FIFO head, copy independence, length and capacity during dynamic growth.</summary>
<description>
Owns a dynamic queue and copied payloads at a stable address. Run from one task.
Teardown clears surviving entries and releases dynamic capacity.
</description>
*)

{attribute 'no_assign'}
{attribute 'no_explicit_call' := 'do not call this function block directly'}
FUNCTION_BLOCK DynamicQueueEnqueueAndPeekTest EXTENDS TOF_Testing.SingleCycleTest
VAR_STAT
	{attribute 'hide'}
	_ClassName : STRING := __POUNAME();
END_VAR
VAR
	_Queue : TOF_Collections.Queue<0>(valueValidator := 0);
END_VAR

(*!
<summary>Checks FIFO head, copy independence, length and capacity during dynamic growth.</summary>
*)
METHOD PROTECTED ExecuteTest
VAR
	values : ARRAY [1..4] OF INT := [11, 22, 33, 44];
END_VAR
_Queue.DefaultDynamicAllocationElementCount := BYTE#2;

_Queue.EnqueueCopy(value := values[1]);
values[1] := 111;

Assert.ThatInt(
	actual := _Queue.Peek().AsInt(),
	message := "Changing the source must preserve the copied head"
).ToBe(expected := INT#11);

Assert.ThatDInt(
	actual := _Queue.Capacity,
	message := "First enqueue must allocate two slots"
).ToBe(expected := DINT#2);

_Queue.EnqueueCopy(value := values[2]);

Assert.ThatInt(
	actual := _Queue.Peek().AsInt(),
	message := "Second enqueue must preserve the head"
).ToBe(expected := INT#11);

Assert.ThatBool(
	actual := _Queue.Full,
	message := "A dynamic queue must report not full when length equals capacity"
).IsFalse();

_Queue.EnqueueCopy(value := values[3]);

Assert.ThatInt(
	actual := _Queue.Peek().AsInt(),
	message := "Growing the descriptor buffer must preserve the head"
).ToBe(expected := INT#11);

Assert.ThatDInt(
	actual := _Queue.Length,
	message := "Three enqueues must produce three entries"
).ToBe(expected := DINT#3);

Assert.ThatDInt(
	actual := _Queue.Capacity,
	message := "Third enqueue must grow to four slots"
).ToBe(expected := DINT#4);

Assert.ThatInt(
	actual := _Queue.GetByIndex(index := 2).AsInt(),
	message := "Third enqueue must append the tail"
).ToBe(expected := values[3]);
END_METHOD

(*!
<summary>Clears the fixture before the runner publishes the result.</summary>
<description>
Also runs after an unexpected exception interrupts the case.
</description>
*)
METHOD PROTECTED AfterTest
_Queue.Clear();
END_METHOD

//! <summary>Borrows the concrete class name. Callers must not modify it.</summary>
{attribute 'monitoring' := 'call'}
PROPERTY ClassName : REFERENCE TO STRING
GET
ClassName REF= _ClassName;
END_GET
END_PROPERTY

//! <summary>Borrows the compiler-initialized namespace name. Callers must not modify it.</summary>
{attribute 'monitoring' := 'call'}
PROPERTY NamespaceName : REFERENCE TO STRING
GET
NamespaceName REF= CurrentNamespace.Name;
END_GET
END_PROPERTY

//! <summary>Reports the concrete instance size in bytes.</summary>
{attribute 'monitoring' := 'call'}
PROPERTY SelfSize : ULINT
GET
SelfSize := XSIZEOF(THIS^);
END_GET
END_PROPERTY

END_FUNCTION_BLOCK

// ---- Tests/Collections/Dynamic/DynamicQueueClearTest.TcPOU
(*
SPDX-FileCopyrightText: c 2026 Oleksandr Tiutyk <trofimich@gmail.com>
SPDX-License-Identifier: MIT
License: https://opensource.org/license/mit
*)

(*!
<summary>Checks release of populated storage and allocation on reuse.</summary>
<description>
Owns a dynamic queue and copied payloads at a stable address. Run from one task.
Teardown clears surviving entries and releases dynamic capacity.
</description>
*)

{attribute 'no_assign'}
{attribute 'no_explicit_call' := 'do not call this function block directly'}
FUNCTION_BLOCK DynamicQueueClearTest EXTENDS TOF_Testing.SingleCycleTest
VAR_STAT
	{attribute 'hide'}
	_ClassName : STRING := __POUNAME();
END_VAR
VAR
	_Queue : TOF_Collections.Queue<0>(valueValidator := 0);
END_VAR

(*!
<summary>Checks release of populated storage and allocation on reuse.</summary>
*)
METHOD PROTECTED ExecuteTest
VAR
	values : ARRAY [1..4] OF INT := [11, 22, 33, 44];
END_VAR
_Queue.DefaultDynamicAllocationElementCount := BYTE#2;

_Queue
	.EnqueueCopy(value := values[1])
	.EnqueueCopy(value := values[2])
	.EnqueueCopy(value := values[3]);

Assert.ThatBool(
	actual := _Queue.Length = 3 AND_THEN _Queue.Capacity = 4,
	message := "The clear fixture must contain three entries in grown storage"
).IsTrue();

_Queue.Clear();

Assert.ThatBool(
	actual := _Queue.Empty AND_THEN _Queue.Length = 0 AND_THEN _Queue.Capacity = 0,
	message := "Clearing a dynamic queue must release its capacity and empty it"
).IsTrue();

Assert.ThatBool(
	actual := _Queue.Contains(value := values[3]),
	message := "Clearing must hide the previous tail"
).IsFalse();

_Queue.Clear();
_Queue.EnqueueCopy(value := values[4]);

Assert.ThatInt(
	actual := _Queue.Peek().AsInt(),
	message := "The cleared queue must accept a fresh head"
).ToBe(expected := values[4]);

Assert.ThatBool(
	actual := _Queue.Length = 1 AND_THEN _Queue.Capacity = 2,
	message := "The fresh head must allocate only the initial capacity"
).IsTrue();
END_METHOD

(*!
<summary>Clears the fixture before the runner publishes the result.</summary>
<description>
Also runs after an unexpected exception interrupts the case.
</description>
*)
METHOD PROTECTED AfterTest
_Queue.Clear();
END_METHOD

//! <summary>Borrows the concrete class name. Callers must not modify it.</summary>
{attribute 'monitoring' := 'call'}
PROPERTY ClassName : REFERENCE TO STRING
GET
ClassName REF= _ClassName;
END_GET
END_PROPERTY

//! <summary>Borrows the compiler-initialized namespace name. Callers must not modify it.</summary>
{attribute 'monitoring' := 'call'}
PROPERTY NamespaceName : REFERENCE TO STRING
GET
NamespaceName REF= CurrentNamespace.Name;
END_GET
END_PROPERTY

//! <summary>Reports the concrete instance size in bytes.</summary>
{attribute 'monitoring' := 'call'}
PROPERTY SelfSize : ULINT
GET
SelfSize := XSIZEOF(THIS^);
END_GET
END_PROPERTY

END_FUNCTION_BLOCK

// ---- Tests/Collections/Dynamic/DynamicQueueRemoveFirstTest.TcPOU
(*
SPDX-FileCopyrightText: c 2026 Oleksandr Tiutyk <trofimich@gmail.com>
SPDX-License-Identifier: MIT
License: https://opensource.org/license/mit
*)

(*!
<summary>Checks FIFO compaction through empty, capacity retention and reuse.</summary>
<description>
Owns a dynamic queue and copied payloads at a stable address. Run from one task.
Teardown clears surviving entries and releases dynamic capacity.
</description>
*)

{attribute 'no_assign'}
{attribute 'no_explicit_call' := 'do not call this function block directly'}
FUNCTION_BLOCK DynamicQueueRemoveFirstTest EXTENDS TOF_Testing.SingleCycleTest
VAR_STAT
	{attribute 'hide'}
	_ClassName : STRING := __POUNAME();
END_VAR
VAR
	_Queue : TOF_Collections.Queue<0>(valueValidator := 0);
END_VAR

(*!
<summary>Checks FIFO compaction through empty, capacity retention and reuse.</summary>
*)
METHOD PROTECTED ExecuteTest
VAR
	values : ARRAY [1..4] OF INT := [11, 22, 33, 44];
END_VAR
_Queue.DefaultDynamicAllocationElementCount := BYTE#2;

_Queue
	.EnqueueCopy(value := values[1])
	.EnqueueCopy(value := values[2])
	.EnqueueCopy(value := values[3]);

_Queue.RemoveFirst();

Assert.ThatInt(
	actual := _Queue.Peek().AsInt(),
	message := "The second entry must become the head after the first removal"
).ToBe(expected := values[2]);

Assert.ThatDInt(
	actual := _Queue.Length,
	message := "Removing the head must leave two entries"
).ToBe(expected := DINT#2);

_Queue.RemoveFirst();

Assert.ThatInt(
	actual := _Queue.Peek().AsInt(),
	message := "The third entry must become the head after the second removal"
).ToBe(expected := values[3]);

_Queue.RemoveFirst();

Assert.ThatBool(
	actual := _Queue.Empty AND_THEN _Queue.Length = 0 AND_THEN _Queue.Capacity = 4,
	message := "Removing the final entry must leave empty storage available for reuse"
).IsTrue();

_Queue.EnqueueCopy(value := values[4]);

Assert.ThatInt(
	actual := _Queue.Peek().AsInt(),
	message := "Reuse after draining must expose the new head"
).ToBe(expected := values[4]);

Assert.ThatDInt(
	actual := _Queue.Capacity,
	message := "Reuse must keep the original capacity until Clear"
).ToBe(expected := DINT#4);
END_METHOD

(*!
<summary>Clears the fixture before the runner publishes the result.</summary>
<description>
Also runs after an unexpected exception interrupts the case.
</description>
*)
METHOD PROTECTED AfterTest
_Queue.Clear();
END_METHOD

//! <summary>Borrows the concrete class name. Callers must not modify it.</summary>
{attribute 'monitoring' := 'call'}
PROPERTY ClassName : REFERENCE TO STRING
GET
ClassName REF= _ClassName;
END_GET
END_PROPERTY

//! <summary>Borrows the compiler-initialized namespace name. Callers must not modify it.</summary>
{attribute 'monitoring' := 'call'}
PROPERTY NamespaceName : REFERENCE TO STRING
GET
NamespaceName REF= CurrentNamespace.Name;
END_GET
END_PROPERTY

//! <summary>Reports the concrete instance size in bytes.</summary>
{attribute 'monitoring' := 'call'}
PROPERTY SelfSize : ULINT
GET
SelfSize := XSIZEOF(THIS^);
END_GET
END_PROPERTY

END_FUNCTION_BLOCK

// ---- Tests/Collections/Dynamic/DynamicDictionaryTestGroup.TcPOU
(*
SPDX-FileCopyrightText: c 2026 Oleksandr Tiutyk <trofimich@gmail.com>
SPDX-License-Identifier: MIT
License: https://opensource.org/license/mit
*)

(*!
<summary>Groups dynamic dictionary lookup, update, removal and clear cases.</summary>
<description>
Owns the child cases, their fixed registration array and the dictionaries borrowed by the common cases.
Each borrowed fixture is reserved for its case throughout the group lifetime. Use from one task at a stable address.
</description>
*)

{attribute 'no_assign'}
{attribute 'no_explicit_call' := 'do not call this function block directly'}
FUNCTION_BLOCK DynamicDictionaryTestGroup EXTENDS TOF_Testing.TestGroup<4>
VAR_STAT
	{attribute 'hide'}
	_ClassName : STRING := __POUNAME();
END_VAR
VAR
	_SetAndGetDictionary : TOF_Collections.Dictionary<0>(keyValidator := 0, valueValidator := 0, keyEqualityComparer := 0);
	_RemoveDictionary : TOF_Collections.Dictionary<0>(keyValidator := 0, valueValidator := 0, keyEqualityComparer := 0);
	_ContainsDictionary : TOF_Collections.Dictionary<0>(keyValidator := 0, valueValidator := 0, keyEqualityComparer := 0);

	_SetAndGet : DictionarySetAndGetTest(name := "SetAndGet", parent := THIS^, dictionary := _SetAndGetDictionary);
	_Remove : DictionaryRemoveTest(name := "Remove", parent := THIS^, dictionary := _RemoveDictionary);
	_Contains : DictionaryContainsTest(name := "Contains", parent := THIS^, dictionary := _ContainsDictionary);
	_Clear : DynamicDictionaryClearTest(name := "Clear", parent := THIS^);

	_Children : ARRAY [0.._ChildCount - 1] OF TOF_Testing.ITestElement :=
	[
		_SetAndGet,
		_Remove,
		_Contains,
		_Clear
	];
END_VAR

//! <summary>Borrows the fixed child array. Callers must not modify it.</summary>
{attribute 'monitoring' := 'call'}
PROPERTY Children : REFERENCE TO ARRAY [0.._ChildCount - 1] OF TOF_Testing.ITestElement
GET
Children REF= _Children;
END_GET
END_PROPERTY

//! <summary>Borrows the concrete class name. Callers must not modify it.</summary>
{attribute 'monitoring' := 'call'}
PROPERTY ClassName : REFERENCE TO STRING
GET
ClassName REF= _ClassName;
END_GET
END_PROPERTY

//! <summary>Borrows the compiler-initialized namespace name. Callers must not modify it.</summary>
{attribute 'monitoring' := 'call'}
PROPERTY NamespaceName : REFERENCE TO STRING
GET
NamespaceName REF= CurrentNamespace.Name;
END_GET
END_PROPERTY

//! <summary>Reports the concrete instance size in bytes.</summary>
{attribute 'monitoring' := 'call'}
PROPERTY SelfSize : ULINT
GET
SelfSize := XSIZEOF(THIS^);
END_GET
END_PROPERTY

END_FUNCTION_BLOCK

// ---- Tests/Collections/DictionarySetAndGetTest.TcPOU
(*
SPDX-FileCopyrightText: c 2026 Oleksandr Tiutyk <trofimich@gmail.com>
SPDX-License-Identifier: MIT
License: https://opensource.org/license/mit
*)

(*!
<summary>Checks updating a stored key, value lookup and indexed retrieval.</summary>
<description>
Borrows one group-owned dictionary reserved for this case. Use from one task at a stable address.
Teardown clears entries owned by the dictionary before publication.
</description>
*)

{attribute 'no_assign'}
{attribute 'no_explicit_call' := 'do not call this function block directly'}
FUNCTION_BLOCK DictionarySetAndGetTest EXTENDS TOF_Testing.SingleCycleTest
VAR_STAT
	{attribute 'hide'}
	_ClassName : STRING := __POUNAME();
END_VAR
VAR
	_Dictionary : TOF_Collections.IDictionary;
	_ReplacementKey : INT := 5;
	_ReplacementValue : STRING := 'Updated5';
END_VAR

(*!
<summary>Binds the dictionary fixture for this case.</summary>
<description>
Stores a borrowed interface without invoking the fixture. The owning group keeps it alive and
reserves it for this case. TestElement initializes the name and parent.
</description>
<param name="name">Display name of this case.</param>
<param name="parent">Group that owns this case.</param>
<param name="dictionary">Required live dictionary reserved for this case.</param>
*)
METHOD FB_init : BOOL
VAR_INPUT
	bInitRetains: BOOL; // TRUE: the retain variables are initialized (reset warm / reset cold)
	bInCopyCode: BOOL; // TRUE: the instance will be copied to the copy code afterward (online change)
	name : WSTRING;
	parent : TOF_Testing.ITestElement;
	dictionary : TOF_Collections.IDictionary;
END_VAR
_Dictionary := dictionary;
FB_init := TRUE;
END_METHOD

(*!
<summary>Checks updating a stored key, value lookup and indexed retrieval.</summary>
*)
METHOD PROTECTED ExecuteTest
VAR
	keys : ARRAY [0..6] OF INT := [0, 1, 2, 3, 4, 5, 6];
	values : ARRAY [0..6] OF STRING :=
		['String0', 'String1', 'String2', 'String3', 'String4', 'String5', 'String6'];
	i : DINT;
	copyReplacement : STRING := 'Updated3';
	position : DINT;
	genericPosition : DINT;
	found : BOOL;

	query : TOF_Core.GENERIC_VALUE;
	value : TOF_Core.GENERIC_VALUE;
	pair : REFERENCE TO TOF_Core.GENERIC_KEY_VALUE_PAIR;
END_VAR
FOR i := 6 TO 0 BY -1 DO
	_Dictionary.SetCopy(key := keys[i], value := values[i]);
END_FOR

_Dictionary.SetCopy(key := keys[3], value := copyReplacement);

query := TOF_Core.GenericValueFactory.FromIntReference(value := _ReplacementKey);
value := TOF_Core.GenericValueFactory.FromStringReference(value := _ReplacementValue);
_Dictionary.SetGeneric(key := query, value := value);

Assert.ThatDInt(
	actual := _Dictionary.Length,
	message := "Updating existing keys must preserve length"
).ToBe(expected := DINT#7);

